(* IEC 61131-3 sources: Industry-PLC-LLM/data/PLCBEAD_repo/PLCBEAD_PLCEmbed-main/PLC-BEAD/Source/OpenPLCv2 (part 6) *)

(* ---- INC_DEC.ST ---- *)
FUNCTION_BLOCK INC_DEC_Block

	VAR_INPUT
		CHA :	BOOL;
		CHB :	BOOL;
		RST :	BOOL := 0;
	END_VAR

	VAR_OUTPUT
		DIR :	BOOL;
		CNT :	INT;
	END_VAR

	VAR
		edgea :	BOOL := 0;
		clk :	BOOL;
		clka :	BOOL;
		clkb :	BOOL;
		edgeb :	BOOL;
		axb :	BOOL;
	END_VAR

	axb := cha XOR chb;

	clka := cha XOR edgea;
	edgea := cha;

	clkb := chb XOR edgeb;
	edgeb := chb;

	clk := clka OR clkb;

	IF axb AND clka THEN dir := TRUE; END_IF;
	IF axb AND clkb THEN dir := FALSE; END_IF;

	IF clk AND dir THEN cnt := cnt + 1; END_IF;
	IF clk AND NOT dir THEN cnt := cnt -1; END_IF;

	IF rst THEN cnt := 0; END_IF;

END_FUNCTION_BLOCK

PROGRAM program0

	VAR
		CHA :	BOOL;
		CHB :	BOOL;
		RST :	BOOL := 0;

		DIR :	BOOL;
		CNT :	INT;
		func_block : INC_DEC_Block;
	END_VAR
	func_block.CHA := CHA;
	func_block.CHB := CHB;
	func_block.RST := RST;
	func_block();
	DIR := func_block.DIR;
	CNT := func_block.CNT;

END_PROGRAM

CONFIGURATION Config0

	RESOURCE Res0 ON PLC
		TASK task0(INTERVAL := T#20ms,PRIORITY := 0);
		PROGRAM instance0 WITH task0 : program0;
	END_RESOURCE

END_CONFIGURATION

(* ---- INSERT250.ST ---- *)
TYPE
	oscat_STRING250             : STRING;
END_TYPE

FUNCTION_BLOCK _INSERT250
    VAR_INPUT
        IN1 :	oscat_STRING250;
        IN2 :	oscat_STRING250;
        P :	INT;
    END_VAR
    VAR_OUTPUT
        _INSERT :	oscat_STRING250;
    END_VAR
    VAR
        size :	INT;
    END_VAR

    size := LEN(IN1);
    IF size + LEN(IN2) <= 250 THEN
        P := LIMIT(0,P,size);
        IF P = 0 THEN
            _INSERT := CONCAT(IN2,IN1);
        ELSE
            _INSERT := INSERT(IN1, IN2, P);
        END_IF;
    END_IF;

END_FUNCTION_BLOCK

PROGRAM program0
	VAR
	    LocalVar1 : oscat_STRING250;
        LocalVar2 : oscat_STRING250;
        LocalVar3 : INT;
		LocalOUT  : oscat_STRING250;
		func_block : _INSERT250;
  	END_VAR
	func_block.IN1 := LocalVar1;
    func_block.IN2 := LocalVar2;
    func_block.P := LocalVar3;
	func_block();
	LocalOUT := func_block._INSERT;
END_PROGRAM

CONFIGURATION Config0
  	RESOURCE Res0 ON PLC
    	TASK task0(INTERVAL := T#20ms,PRIORITY := 0);
    	PROGRAM instance0 WITH task0 : program0;
  	END_RESOURCE
END_CONFIGURATION

(* ---- INTEGRATE.ST ---- *)
FUNCTION_BLOCK T_PLC_MS_block
	VAR_OUTPUT
		T_PLC_MS :	UDINT;
	END_VAR

	VAR_EXTERNAL
		PLC_TICKS_PER_SEC :	INT;
		PLC_SYS_TICK_CNT :	DINT;
	END_VAR

	VAR
		debug :	BOOL;(*Debug-Mode ON / OFF*)
		N :	INT;(*Debug-Faktor*)
		Offset :	UDINT;(*Debug-Offset*)
		temp :	DWORD := DWORD#1;(*Debug-Offset*)
		mode :	BOOL;(*modus*)
		faktor :	UDINT;(*Systemtakt-Faktor*)
		init :	BOOL;
		v_plc_ticks_per_sec :	UDINT;
		base :	UDINT := UDINT#1000;
	END_VAR

	IF init = FALSE THEN
		v_plc_ticks_per_sec := INT_TO_UDINT(PLC_TICKS_PER_SEC);
		IF v_plc_ticks_per_sec = UDINT#1024 THEN
			faktor := UDINT#1;
			mode := FALSE;
		ELSIF v_plc_ticks_per_sec > UDINT#0 THEN
			IF v_plc_ticks_per_sec <= base THEN
				faktor := base / v_plc_ticks_per_sec;
				mode := FALSE;
			ELSE
				faktor := v_plc_ticks_per_sec / base;
				mode := TRUE;
			END_IF;
		ELSE
			faktor := UDINT#1;
		END_IF;
		init := TRUE;
	END_IF;

	IF mode THEN
		T_PLC_MS := DINT_TO_UDINT(PLC_SYS_TICK_CNT) / faktor;
	ELSE
		T_PLC_MS := DINT_TO_UDINT(PLC_SYS_TICK_CNT) * faktor;
	END_IF;

	IF debug THEN
		T_PLC_MS := (DWORD_TO_UDINT(SHL(UDINT_TO_DWORD(T_PLC_MS),N) OR SHL(temp,N)) - UDINT#1) + Offset;
	END_IF;
END_FUNCTION_BLOCK

FUNCTION_BLOCK INTEGRATE

	VAR_INPUT
		E :	BOOL := TRUE;
		X :	REAL;
		K :	REAL := 1.0;
	END_VAR

	VAR_IN_OUT
		Y :	REAL;
	END_VAR

	VAR
		X_last :	REAL;
		init :	BOOL;
		T_PLC_MS :	T_PLC_MS_block;
		last :	UDINT;
		tx :	UDINT;
	END_VAR

	T_PLC_MS();
	tx:= T_PLC_MS.T_PLC_MS;

	IF NOT init THEN
		init := TRUE;
		X_last := X;
	ELSIF E THEN
		Y := (X + X_LAST) * 0.5E-3 * UDINT_TO_REAL(tx-last) * K + Y;
		X_last := X;
	END_IF;
	last := tx;

END_FUNCTION_BLOCK

PROGRAM program0
  VAR
	E :	BOOL := TRUE;
	X :	REAL;
	K :	REAL := 1.0;

	Y :	REAL;

	func_block : INTEGRATE;
  END_VAR
	func_block.E:=E;
	func_block.X:=X;
	func_block.K:=K;
	func_block.Y:=Y;
	func_block();
	Y:= func_block.Y;
END_PROGRAM

CONFIGURATION Config0
	VAR_GLOBAL
		PLC_TICKS_PER_SEC :	INT;
		PLC_SYS_TICK_CNT :	DINT;
	END_VAR
	RESOURCE Res0 ON PLC
		TASK task0(INTERVAL := T#20ms,PRIORITY := 0);
		PROGRAM instance0 WITH task0 : program0;
	END_RESOURCE
END_CONFIGURATION

(* ---- INTERLOCK.ST ---- *)
FUNCTION_BLOCK INTERLOCK_Block

	VAR_INPUT
		I1 :	BOOL;
		I2 :	BOOL;
		TL :	TIME;
	END_VAR

	VAR_OUTPUT
		Q1 :	BOOL;
		Q2 :	BOOL;
	END_VAR

	VAR
		T1 :	TOF;
		T2 :	TOF;
	END_VAR

	T1(IN := I1, PT := TL);
	T2(IN := I2, PT := TL);

	Q1 := I1 AND NOT t2.Q;
	Q2 := I2 AND NOT t1.Q;

END_FUNCTION_BLOCK

PROGRAM program0
	VAR
		I1 :	BOOL;
		I2 :	BOOL;
		TL :	TIME;
		Q1 :	BOOL;
		Q2 :	BOOL;
		func_block : INTERLOCK_Block;
  	END_VAR
	func_block.I1  :=I1;
	func_block.I2  :=I2;
	func_block.TL  :=TL;
	func_block();
	Q1 := func_block.Q1;
	Q2 := func_block.Q2;
END_PROGRAM

CONFIGURATION Config0
	RESOURCE Res0 ON PLC
		TASK task0(INTERVAL := T#20ms,PRIORITY := 0);
		PROGRAM instance0 WITH task0 : program0;
	END_RESOURCE
END_CONFIGURATION

(* ---- INTERLOCK_4.ST ---- *)
FUNCTION BIT_LOAD_B:BYTE
	VAR_INPUT
		IN :	BYTE;
		VAL :	BOOL;
		POS :	INT;
	END_VAR

	IF VAL THEN
		BIT_LOAD_B := in OR SHL(BYTE#1,pos);
	ELSE
		BIT_LOAD_B := in AND (NOT SHL(BYTE#1,pos));
	END_IF;
END_FUNCTION

FUNCTION_BLOCK INTERLOCK_4_Block

	VAR_INPUT
		I0 :	BOOL;
		I1 :	BOOL;
		I2 :	BOOL;
		I3 :	BOOL;
		E :	BOOL;
		MODE :	INT;
	END_VAR

	VAR_OUTPUT
		OUT :	BYTE;
		_TP :	BOOL;
	END_VAR

	VAR
		in :	BYTE;
		last :	BYTE;
		old :	BYTE;
		lmode :	INT;
	END_VAR

	IF E THEN
	(* reset all vars when there is a mode change on thy fly *)
		IF mode <> lmode THEN
			out := BYTE#0;
			last := BYTE#0;
			old := BYTE#0;
			lmode := mode;
		END_IF;
		(* load inputs into in *)
		in:=BIT_LOAD_B(in,I0,0); (* in.0 *)
		in:=BIT_LOAD_B(in,I1,1); (* in.1 *)
		in:=BIT_LOAD_B(in,I2,2); (* in.2 *)
		in:=BIT_LOAD_B(in,I3,3); (* in.3 *)
		(* only execute when there is any change *)
		IF in <> last THEN
			(* only execute when inputs have chages state *)
			CASE mode OF
				0:	(* output directly display inputs as bits in byte out *)
					out := in;

				1:	(* the input with the highest number will be acepted *)
					IF    (in AND BYTE#2#00001000) > BYTE#0 (* in.3 *) THEN out := BYTE#8;
					ELSIF (in AND BYTE#2#00000100) > BYTE#0 (* in.2 *) THEN out := BYTE#4;
					ELSIF (in AND BYTE#2#00000010) > BYTE#0 (* in.1 *) THEN out := BYTE#2;
					ELSE out := in;
					END_IF;

				2:	(* input last pressed will be displayed only *)
					last := ((in XOR last) AND in);
					IF    (last AND BYTE#2#00001000) > BYTE#0 (* last.3 *) THEN out := BYTE#8;
					ELSIF (last AND BYTE#2#00000100) > BYTE#0 (* last.2 *) THEN out := BYTE#4;
					ELSIF (last AND BYTE#2#00000010) > BYTE#0 (* last.1 *) THEN out := BYTE#2;
					ELSE out := last;
					END_IF;

				3:	(* any input active will disable all other inputs *)
					IF (out AND in) = BYTE#0 THEN
						IF    (in AND BYTE#2#00001000) > BYTE#0 (* in.3 *) THEN out := BYTE#8;
						ELSIF (in AND BYTE#2#00000100) > BYTE#0 (* in.2 *) THEN out := BYTE#4;
						ELSIF (in AND BYTE#2#00000010) > BYTE#0 (* in.1 *) THEN out := BYTE#2;
						ELSE out := in;
						END_IF;
					END_IF;

			END_CASE;
			last := in;
		END_IF;
		_tp := out <> old;
		old := out;
	ELSE
		out := BYTE#0;
		last := BYTE#0;
		old := BYTE#0;
		lmode := 0;
		_tp := FALSE;
	END_IF;

END_FUNCTION_BLOCK

PROGRAM program0

	VAR
		I0 :	BOOL;
		I1 :	BOOL;
		I2 :	BOOL;
		I3 :	BOOL;
		E :	BOOL;
		MODE :	INT;
		OUT :	BYTE;
		_TP :	BOOL;
		func_block : INTERLOCK_4_Block;
	END_VAR
	func_block.I0 := I0;
	func_block.I1 := I1;
	func_block.I2 := I2;
	func_block.I3 := I3;
	func_block.E := E;
	func_block.MODE := MODE;
	func_block();
	OUT := func_block.OUT;
	_TP := func_block._TP;

END_PROGRAM

CONFIGURATION Config0

	RESOURCE Res0 ON PLC
		TASK task0(INTERVAL := T#20ms,PRIORITY := 0);
		PROGRAM instance0 WITH task0 : program0;
	END_RESOURCE

END_CONFIGURATION

(* ---- IP4_TO_STRING.ST ---- *)
TYPE
  oscat_STRING10             : STRING;
END_TYPE

FUNCTION _BYTE_TO_INT:INT
	VAR_INPUT
		IN :	BYTE;
	END_VAR

	_BYTE_TO_INT := USINT_TO_INT(BYTE_TO_USINT(IN));
END_FUNCTION

FUNCTION BYTE_OF_DWORD:BYTE
	VAR_INPUT
		IN :	DWORD;
		N :	BYTE;
	END_VAR
	BYTE_OF_DWORD := DWORD_TO_BYTE(SHR(in,_BYTE_TO_INT(SHL(n,3))));
END_FUNCTION

FUNCTION_BLOCK IP4_TO_STRING_Block

	VAR_INPUT
		IP4 :	DWORD;
	END_VAR

	VAR_OUTPUT
		IP4_TO_STRING :	STRING;
	END_VAR

	VAR
		s1 :	oscat_string10;
		s2 :	oscat_string10;
	END_VAR

	s1 := CONCAT(BYTE_TO_STRING(BYTE_OF_DWORD(IP4,BYTE#1)),BYTE_TO_STRING(BYTE_OF_DWORD(IP4,BYTE#0)));
	s2 := CONCAT(BYTE_TO_STRING(BYTE_OF_DWORD(IP4,BYTE#3)),BYTE_TO_STRING(BYTE_OF_DWORD(IP4,BYTE#2)));
	IP4_TO_STRING := CONCAT(s2,s1);

END_FUNCTION_BLOCK

PROGRAM program0
	VAR
		IP4 :	DWORD;
		IP4_TO_STRING :	STRING;

		func_block : IP4_TO_STRING_Block;
	END_VAR
	func_block.IP4 := IP4;

	func_block();
	IP4_TO_STRING  := func_block.IP4_TO_STRING;
END_PROGRAM

CONFIGURATION Config0

  	RESOURCE Res0 ON PLC
    	TASK task0(INTERVAL := T#20ms,PRIORITY := 0);
    	PROGRAM instance0 WITH task0 : program0;
  	END_RESOURCE

END_CONFIGURATION

(* ---- IRTRANS_DECODE.ST ---- *)
FUNCTION_BLOCK CHR_TO_STRING_Block
	VAR_INPUT
		C :	BYTE;
	END_VAR

	VAR_OUTPUT
		CHR_TO_STRING :	STRING;
	END_VAR

	CHR_TO_STRING := BYTE_TO_STRING(C);

END_FUNCTION_BLOCK

TYPE

  oscat_NW_BUF_SHORT : ARRAY [0..1407] OF BYTE;
  oscat_NW_BUF_LONG  : ARRAY [0..4095] OF BYTE;

  oscat_NETWORK_BUFFER_SHORT :
  STRUCT
    SIZE   : UINT;
    BUFFER : oscat_NW_BUF_SHORT;
  END_STRUCT;

  oscat_NETWORK_BUFFER :
  STRUCT
    SIZE   : UINT;
    BUFFER : oscat_NW_BUF_LONG;
  END_STRUCT;

END_TYPE

TYPE
  oscat_IP_FIFO128_DATA  : ARRAY [1..128] OF BYTE;
  oscat_Mailbox  : ARRAY [1..16] OF BYTE;

  oscat_IP_FIFO_DATA :
  STRUCT
	X       : oscat_IP_FIFO128_DATA; (* IP_ID FIFO Speicher          *)
	Y       : oscat_IP_FIFO128_DATA; (* IP_ID Z�hler                 *)
	ID      : BYTE;                  (* h�chste vergabene id         *)
	MAX_ID  : BYTE;                  (* maximal Anmeldungen pro ID   *)
    INIT    : BOOL;                  (* Initialisierung durchgef�hrt *)
	EMPTY   : BOOL;                  (* FIFO leer                    *)
	FULL    : BOOL;                  (* FIFO voll                    *)
	TOP     : INT;                   (* maximale anzahl in FIFO      *)
	NW      : INT;                   (* Schreibzeiger                *)
	NR      : INT;                   (* Lesezeiger                   *)
  END_STRUCT;

  oscat_IP_C:
  STRUCT
  	C_MODE:			BYTE;          		(*W Mode: TCP/UCP AKTIV/PASSIV                               *)
	C_PORT:         WORD;          		(*W Portnummer                                               *)
	C_IP:           DWORD;         		(*W IP-Adresse gepackt wwxxyyzz = www.xxx.yyy.zzz            *)
    C_STATE:        BYTE;          		(*R Verbindungsstatus ON/OFF + Flanke ON/OFF                 *)
	C_ENABLE:       BOOL;          		(*W Freigabe f�r Connect                                     *)
    R_OBSERVE:      BOOL;          		(*W Empfang ueberwachen                                      *)
    TIME_RESET:     BOOL;          		(*W Alle Timer ruecksetzen                                   *)
	ERROR:          DWORD;         		(*R vvwwxxyy (vv = CON_ERROR, ww = SEN_ERROR, xx = REC_ERROR *)
    FIFO:           oscat_IP_FIFO_DATA; (*I IP FIFO Struktur                                         *)
	MAILBOX:		oscat_Mailbox;		(*I Mailbox: Datenbereich f�r Bausteindatenaustausch         *)
  END_STRUCT;
END_TYPE

FUNCTION_BLOCK IRTRANS_DECODE_Block

	VAR_OUTPUT
		CMD :	BOOL;
		DEV :	STRING;
		KEY :	STRING;
		ERROR :	BOOL;
	END_VAR

	VAR_IN_OUT
		IP_C :	oscat_IP_C;
		R_BUF :	oscat_NETWORK_BUFFER;
	END_VAR

	VAR
		i :	INT;
		stop :	INT;
		received_string :	STRING;
		char :	STRING;
		CHR_TO_STRING :	CHR_TO_STRING_Block;
		z :	BYTE;
	END_VAR

	i := UINT_TO_INT(R_BUF.SIZE);
	IF i >= 5 AND (i <= 82) AND IP_C.MAILBOX[1] <> z THEN
		error := TRUE;
		i := i - 1;

		IF R_BUF.BUFFER[i] <> BYTE#10 THEN RETURN; END_IF;
		i := i - 1;
		IF R_BUF.BUFFER[i] <> BYTE#13 THEN RETURN; END_IF;
		i := i - 1;

		stop := 0;
		received_string := '';

		WHILE stop <= i DO
			CHR_TO_STRING(C:=R_BUF.BUFFER[stop]);
			char := CHR_TO_STRING.CHR_TO_STRING;
			received_string := CONCAT(received_string,char);
			stop := stop + INT#1;
		END_WHILE;

		stop := FIND(received_string,',');
		IF stop > 0 AND stop - 1 < i THEN
			DEV := LEFT(received_string,stop - 1);
			key := RIGHT(received_string,i - stop + 1);
			IF LEN(DEV) = 0 OR LEN(key) = 0 THEN RETURN; END_IF;
			cmd := TRUE;
			error := FALSE;
		END_IF;
	ELSE
		cmd := FALSE;
		error := FALSE;
	END_IF;

	z := IP_C.MAILBOX[1];

END_FUNCTION_BLOCK

PROGRAM program0
	VAR
		IP_C :	oscat_IP_C;
		R_BUF :	oscat_NETWORK_BUFFER;
		CMD :	BOOL;
		DEV :	STRING;
		KEY :	STRING;
		ERROR :	BOOL;

		func_block : IRTRANS_DECODE_Block;
	END_VAR
	func_block.IP_C := IP_C;
	func_block.R_BUF := R_BUF;

	func_block();
	IP_C  := func_block.IP_C;
	R_BUF  := func_block.R_BUF;
	CMD  := func_block.CMD;
	DEV  := func_block.DEV;
	KEY  := func_block.KEY;
	ERROR  := func_block.ERROR;

END_PROGRAM

CONFIGURATION Config0

  	RESOURCE Res0 ON PLC
    	TASK task0(INTERVAL := T#20ms,PRIORITY := 0);
    	PROGRAM instance0 WITH task0 : program0;
  	END_RESOURCE

END_CONFIGURATION

(* ---- IRTRANS_RCV_1.ST ---- *)
FUNCTION_BLOCK IRTRANS_RCV_1_Block

	VAR_INPUT
		CMD :	BOOL;
		DEV_CODE :	STRING;
		KEY_CODE :	STRING;
	END_VAR

	VAR_OUTPUT
		Q :	BOOL;
	END_VAR

	VAR_IN_OUT
		DEV :	STRING;
		KEY :	STRING;
	END_VAR

	Q := cmd AND EQ_STRING(dev_code,dev) AND EQ_STRING(key_code,key);

END_FUNCTION_BLOCK

PROGRAM program0
	VAR
		CMD :	BOOL;
		DEV :	STRING;
		KEY :	STRING;
		DEV_CODE :	STRING;
		KEY_CODE :	STRING;
		Q :	BOOL;

		func_block : IRTRANS_RCV_1_Block;
	END_VAR
	func_block.CMD := CMD;
	func_block.DEV := DEV;
	func_block.KEY := KEY;
	func_block.DEV_CODE := DEV_CODE;
	func_block.KEY_CODE := KEY_CODE;

	func_block();
	DEV  := func_block.DEV;
	KEY  := func_block.KEY;
	Q  := func_block.Q;

END_PROGRAM

CONFIGURATION Config0

  	RESOURCE Res0 ON PLC
    	TASK task0(INTERVAL := T#20ms,PRIORITY := 0);
    	PROGRAM instance0 WITH task0 : program0;
  	END_RESOURCE

END_CONFIGURATION

(* ---- IRTRANS_RCV_4.ST ---- *)
FUNCTION_BLOCK IRTRANS_RCV_4_Block

	VAR_INPUT
		CMD :	BOOL;
	END_VAR

	VAR_IN_OUT
		DEV :	STRING;
		KEY :	STRING;
	END_VAR

	VAR_INPUT
		DEV_CODE :	STRING;
		KEY_CODE_0 :	STRING;
		KEY_CODE_1 :	STRING;
		KEY_CODE_2 :	STRING;
		KEY_CODE_3 :	STRING;
	END_VAR

	VAR_OUTPUT
		Q0 :	BOOL;
		Q1 :	BOOL;
		Q2 :	BOOL;
		Q3 :	BOOL;
	END_VAR

	VAR
		decode :	BOOL;
	END_VAR

	decode := cmd AND EQ_STRING(dev_code,dev);

	Q0 := EQ_STRING(key,key_code_0) AND decode;
	Q1 := EQ_STRING(key,key_code_1) AND decode;
	Q2 := EQ_STRING(key,key_code_2) AND decode;
	Q3 := EQ_STRING(key,key_code_3) AND decode;

END_FUNCTION_BLOCK

PROGRAM program0
	VAR
		CMD :	BOOL;
		DEV :	STRING;
		KEY :	STRING;
		DEV_CODE :	STRING;
		KEY_CODE_0 :	STRING;
		KEY_CODE_1 :	STRING;
		KEY_CODE_2 :	STRING;
		KEY_CODE_3 :	STRING;
		Q0 :	BOOL;
		Q1 :	BOOL;
		Q2 :	BOOL;
		Q3 :	BOOL;

		func_block : IRTRANS_RCV_4_Block;
	END_VAR
	func_block.CMD := CMD;
	func_block.DEV := DEV;
	func_block.KEY := KEY;
	func_block.DEV_CODE := DEV_CODE;
	func_block.KEY_CODE_0 := KEY_CODE_0;
	func_block.KEY_CODE_1 := KEY_CODE_1;
	func_block.KEY_CODE_2 := KEY_CODE_2;
	func_block.KEY_CODE_3 := KEY_CODE_3;

	func_block();
	DEV  := func_block.DEV;
	KEY  := func_block.KEY;
	Q0  := func_block.Q0;
	Q1  := func_block.Q1;
	Q2  := func_block.Q2;
	Q3  := func_block.Q3;

END_PROGRAM

CONFIGURATION Config0

  	RESOURCE Res0 ON PLC
    	TASK task0(INTERVAL := T#20ms,PRIORITY := 0);
    	PROGRAM instance0 WITH task0 : program0;
  	END_RESOURCE

END_CONFIGURATION

(* ---- IRTRANS_RCV_8.ST ---- *)
FUNCTION_BLOCK IRTRANS_RCV_8_Block

	VAR_INPUT
		CMD :	BOOL;
	END_VAR

	VAR_IN_OUT
		DEV :	STRING;
		KEY :	STRING;
	END_VAR

	VAR_INPUT
		DEV_CODE :	STRING;
		KEY_CODE_0 :	STRING;
		KEY_CODE_1 :	STRING;
		KEY_CODE_2 :	STRING;
		KEY_CODE_3 :	STRING;
		KEY_CODE_4 :	STRING;
		KEY_CODE_5 :	STRING;
		KEY_CODE_6 :	STRING;
		KEY_CODE_7 :	STRING;
	END_VAR

	VAR_OUTPUT
		Q0 :	BOOL;
		Q1 :	BOOL;
		Q2 :	BOOL;
		Q3 :	BOOL;
		Q4 :	BOOL;
		Q5 :	BOOL;
		Q6 :	BOOL;
		Q7 :	BOOL;
	END_VAR

	VAR
		decode :	BOOL;
	END_VAR

	decode := cmd AND EQ_STRING(dev_code,dev);

	Q0 := EQ_STRING(key,key_code_0) AND decode;
	Q1 := EQ_STRING(key,key_code_1) AND decode;
	Q2 := EQ_STRING(key,key_code_2) AND decode;
	Q3 := EQ_STRING(key,key_code_3) AND decode;
	Q4 := EQ_STRING(key,key_code_4) AND decode;
	Q5 := EQ_STRING(key,key_code_5) AND decode;
	Q6 := EQ_STRING(key,key_code_6) AND decode;
	Q7 := EQ_STRING(key,key_code_7) AND decode;

END_FUNCTION_BLOCK

PROGRAM program0
	VAR
		CMD :	BOOL;
		DEV :	STRING;
		KEY :	STRING;
		DEV_CODE :	STRING;
		KEY_CODE_0 :	STRING;
		KEY_CODE_1 :	STRING;
		KEY_CODE_2 :	STRING;
		KEY_CODE_3 :	STRING;
		KEY_CODE_4 :	STRING;
		KEY_CODE_5 :	STRING;
		KEY_CODE_6 :	STRING;
		KEY_CODE_7 :	STRING;
		Q0 :	BOOL;
		Q1 :	BOOL;
		Q2 :	BOOL;
		Q3 :	BOOL;
		Q4 :	BOOL;
		Q5 :	BOOL;
		Q6 :	BOOL;
		Q7 :	BOOL;

		func_block : IRTRANS_RCV_8_Block;
	END_VAR
	func_block.CMD := CMD;
	func_block.DEV := DEV;
	func_block.KEY := KEY;
	func_block.DEV_CODE := DEV_CODE;
	func_block.KEY_CODE_0 := KEY_CODE_0;
	func_block.KEY_CODE_1 := KEY_CODE_1;
	func_block.KEY_CODE_2 := KEY_CODE_2;
	func_block.KEY_CODE_3 := KEY_CODE_3;
	func_block.KEY_CODE_4 := KEY_CODE_4;
	func_block.KEY_CODE_5 := KEY_CODE_5;
	func_block.KEY_CODE_6 := KEY_CODE_6;
	func_block.KEY_CODE_7 := KEY_CODE_7;

	func_block();
	DEV  := func_block.DEV;
	KEY  := func_block.KEY;
	Q0  := func_block.Q0;
	Q1  := func_block.Q1;
	Q2  := func_block.Q2;
	Q3  := func_block.Q3;
	Q4  := func_block.Q4;
	Q5  := func_block.Q5;
	Q6  := func_block.Q6;
	Q7  := func_block.Q7;

END_PROGRAM

CONFIGURATION Config0

  	RESOURCE Res0 ON PLC
    	TASK task0(INTERVAL := T#20ms,PRIORITY := 0);
    	PROGRAM instance0 WITH task0 : program0;
  	END_RESOURCE

END_CONFIGURATION

(* ---- IRTRANS_SERVER.ST ---- *)
TYPE

  oscat_NW_BUF_SHORT : ARRAY [0..1407] OF BYTE;
  oscat_NW_BUF_LONG  : ARRAY [0..4095] OF BYTE;

  oscat_NETWORK_BUFFER_SHORT :
  STRUCT
    SIZE   : UINT;
    BUFFER : oscat_NW_BUF_SHORT;
  END_STRUCT;

  oscat_NETWORK_BUFFER :
  STRUCT
    SIZE   : UINT;
    BUFFER : oscat_NW_BUF_LONG;
  END_STRUCT;

END_TYPE

TYPE
  oscat_IP_FIFO128_DATA  : ARRAY [1..128] OF BYTE;
  oscat_Mailbox  : ARRAY [1..16] OF BYTE;

  oscat_IP_FIFO_DATA :
  STRUCT
	X       : oscat_IP_FIFO128_DATA; (* IP_ID FIFO Speicher          *)
	Y       : oscat_IP_FIFO128_DATA; (* IP_ID Z�hler                 *)
	ID      : BYTE;                  (* h�chste vergabene id         *)
	MAX_ID  : BYTE;                  (* maximal Anmeldungen pro ID   *)
    INIT    : BOOL;                  (* Initialisierung durchgef�hrt *)
	EMPTY   : BOOL;                  (* FIFO leer                    *)
	FULL    : BOOL;                  (* FIFO voll                    *)
	TOP     : INT;                   (* maximale anzahl in FIFO      *)
	NW      : INT;                   (* Schreibzeiger                *)
	NR      : INT;                   (* Lesezeiger                   *)
  END_STRUCT;

  oscat_IP_C:
  STRUCT
  	C_MODE:			BYTE;          		(*W Mode: TCP/UCP AKTIV/PASSIV                               *)
	C_PORT:         WORD;          		(*W Portnummer                                               *)
	C_IP:           DWORD;         		(*W IP-Adresse gepackt wwxxyyzz = www.xxx.yyy.zzz            *)
    C_STATE:        BYTE;          		(*R Verbindungsstatus ON/OFF + Flanke ON/OFF                 *)
	C_ENABLE:       BOOL;          		(*W Freigabe f�r Connect                                     *)
    R_OBSERVE:      BOOL;          		(*W Empfang ueberwachen                                      *)
    TIME_RESET:     BOOL;          		(*W Alle Timer ruecksetzen                                   *)
	ERROR:          DWORD;         		(*R vvwwxxyy (vv = CON_ERROR, ww = SEN_ERROR, xx = REC_ERROR *)
    FIFO:           oscat_IP_FIFO_DATA; (*I IP FIFO Struktur                                         *)
	MAILBOX:		oscat_Mailbox;		(*I Mailbox: Datenbereich f�r Bausteindatenaustausch         *)
  END_STRUCT;
END_TYPE

FUNCTION_BLOCK IRTRANS_SERVER_Block

	VAR_INPUT
		UDP_TCP :	BOOL;
	END_VAR

	VAR_OUTPUT
		S_ENABLE :	BOOL;
		R_ENABLE :	BOOL;
		ERROR :	DWORD;
	END_VAR

	VAR_IN_OUT
		IP_C :	oscat_IP_C;
		S_BUF :	oscat_NETWORK_BUFFER;
		R_BUF :	oscat_NETWORK_BUFFER;
	END_VAR

	VAR
		t :	TON;
	END_VAR

	IF NOT IP_C.C_ENABLE THEN
		IP_C.C_PORT := WORD#0;
		IP_C.C_IP := DWORD#00;
		IP_C.C_MODE := SEL(UDP_TCP,BYTE#5,BYTE#4);
		IP_C.C_ENABLE := TRUE;
		IP_C.R_OBSERVE := FALSE;
		IP_C.TIME_RESET := TRUE;
		S_BUF.SIZE := UINT#0;
		R_BUF.SIZE := UINT#0;
	END_IF;

	R_ENABLE := IP_C.C_STATE > BYTE#127;
	S_ENABLE := R_ENABLE AND (IP_C.MAILBOX[1] > BYTE#0 OR IP_C.C_MODE <> BYTE#5);
	ERROR := IP_C.ERROR;

	t(IN:= IP_C.ERROR > DWORD#0, PT:=T#5s);
	IF t.Q THEN
		IP_C.TIME_RESET := TRUE;
	END_IF;

END_FUNCTION_BLOCK

PROGRAM program0
	VAR
		UDP_TCP :	BOOL;
		S_ENABLE :	BOOL;
		R_ENABLE :	BOOL;
		ERROR :	DWORD;
		IP_C :	oscat_IP_C;
		S_BUF :	oscat_NETWORK_BUFFER;
		R_BUF :	oscat_NETWORK_BUFFER;

		func_block : IRTRANS_SERVER_Block;
	END_VAR
	func_block.UDP_TCP := UDP_TCP;
	func_block.IP_C := IP_C;
	func_block.S_BUF := S_BUF;
	func_block.R_BUF := R_BUF;

	func_block();
	S_ENABLE  := func_block.S_ENABLE;
	R_ENABLE  := func_block.R_ENABLE;
	ERROR  := func_block.ERROR;
	IP_C  := func_block.IP_C;
	S_BUF  := func_block.S_BUF;
	R_BUF  := func_block.R_BUF;

END_PROGRAM

CONFIGURATION Config0

  	RESOURCE Res0 ON PLC
    	TASK task0(INTERVAL := T#20ms,PRIORITY := 0);
    	PROGRAM instance0 WITH task0 : program0;
  	END_RESOURCE

END_CONFIGURATION

(* ---- IS_CC.ST ---- *)
FUNCTION_BLOCK IS_CC_Block

	VAR_INPUT
		STR :	STRING;
		CMP :	STRING;
	END_VAR

	VAR_OUTPUT
		IS_CC :	BOOL;
	END_VAR

	VAR
		L :	INT;
		pos :	INT;
		temp :	STRING;
	END_VAR

	L := LEN(str);
	FOR pos := 1 TO L DO
		temp := MID(str,1,pos);
		IF FIND(CMP,temp) = 0 THEN
			IS_CC := FALSE;
			RETURN;
		END_IF;
	END_FOR;
	IS_CC := L > 0;

END_FUNCTION_BLOCK

PROGRAM program0

	VAR
		STR :	STRING;
		CMP :	STRING;

		IS_CC :	BOOL;

		func_block : IS_CC_Block;
	END_VAR
	func_block.STR := STR;
	func_block.CMP := CMP;
	func_block();
	IS_CC := func_block.IS_CC;

END_PROGRAM

CONFIGURATION Config0

	RESOURCE Res0 ON PLC
		TASK task0(INTERVAL := T#20ms,PRIORITY := 0);
		PROGRAM instance0 WITH task0 : program0;
	END_RESOURCE

END_CONFIGURATION

(* ---- IS_NCC.ST ---- *)
FUNCTION_BLOCK IS_NCC_Block

	VAR_INPUT
		STR :	STRING;
		CMP :	STRING;
	END_VAR

	VAR_OUTPUT
		IS_NCC :	BOOL;
	END_VAR

	VAR
		L :	INT;
		pos :	INT;
		temp :	STRING;
	END_VAR

	L := LEN(str);
	FOR pos := 1 TO L DO
		temp := MID(str,1,pos);
		IF FIND(CMP,temp) > 0 THEN
			IS_NCC := FALSE;
			RETURN;
		END_IF;
	END_FOR;
	IS_NCC := TRUE;

END_FUNCTION_BLOCK

PROGRAM program0

	VAR
		STR :	STRING;
		CMP :	STRING;
		IS_NCC :	BOOL;
		func_block : IS_NCC_Block;
	END_VAR
	func_block.STR := STR;
	func_block.CMP := CMP;
	func_block();
	IS_NCC := func_block.IS_NCC;

END_PROGRAM

CONFIGURATION Config0

	RESOURCE Res0 ON PLC
		TASK task0(INTERVAL := T#20ms,PRIORITY := 0);
		PROGRAM instance0 WITH task0 : program0;
	END_RESOURCE

END_CONFIGURATION

(* ---- IS_SORTED.ST ---- *)
TYPE
	oscat_pt_ARRAY: ARRAY [1..100] OF REAL;
END_TYPE

FUNCTION_BLOCK IS_SORTED_Block

	VAR_IN_OUT
		PT :	oscat_pt_ARRAY;
	END_VAR

	VAR_INPUT
		SIZE :	UINT;
	END_VAR

	VAR_OUTPUT
		IS_SORTED :	BOOL;
	END_VAR

	VAR
		i :	INT;
		i2 :	INT;
		stop :	INT;
	END_VAR

	stop :=LIMIT_INT(1,UINT_TO_INT(size),1000);
	stop := stop -1;
	FOR i := 1 TO stop DO
		i2 := i+1;
		IF pt[i] > pt[i2] THEN
			IS_SORTED := FALSE;
			RETURN;
		END_IF;
	END_FOR;

	IS_SORTED := TRUE;

END_FUNCTION_BLOCK

PROGRAM program0

	VAR
		SIZE :	UINT;
		PT :	oscat_pt_ARRAY;
		IS_SORTED :	BOOL;
		func_block : IS_SORTED_Block;
	END_VAR
	func_block.SIZE := SIZE;
	func_block.PT := PT;
	func_block();
	PT := func_block.PT;
	IS_SORTED := func_block.IS_SORTED;

END_PROGRAM

CONFIGURATION Config0

	RESOURCE Res0 ON PLC
		TASK task0(INTERVAL := T#20ms,PRIORITY := 0);
		PROGRAM instance0 WITH task0 : program0;
	END_RESOURCE

END_CONFIGURATION

(* ---- LAMBERT_W.ST ---- *)
FUNCTION _REAL_TO_DWORD: DWORD

  VAR_INPUT
    X :	REAL;
  END_VAR

  IF REAL_TO_DWORD(0.5) = DWORD#1 THEN
    _REAL_TO_DWORD := REAL_TO_DWORD(x);
  ELSIF X > 0.0 THEN
    _REAL_TO_DWORD := REAL_TO_DWORD(x+0.5);
  ELSIF X < 0.0 THEN
    _REAL_TO_DWORD := REAL_TO_DWORD(x-0.5);
  ELSE
    _REAL_TO_DWORD := DWORD#0;
  END_IF;
END_FUNCTION

FUNCTION_BLOCK LAMBERT_W_Block

	VAR_INPUT
		X :	REAL;
	END_VAR

	VAR_OUTPUT
		LAMBERT_W :	REAL;
	END_VAR

	VAR
		w :	REAL;
		i :	INT;
		we :	REAL;
		w1e :	REAL;
		last :	DWORD;
		ewx :	REAL;
	END_VAR

	IF x < -0.367879441171442 THEN
		LAMBERT_W := -1000.0;
		RETURN;
	(* return 0 if x = 0 *)
	ELSIF x = 0.0 THEN
		RETURN;
	(* first an estimate is calculated *)
	ELSIF x <= 500.0 THEN
		w := LN(x + 1.0);
		w := 0.665 * (1.0 + 0.0195 * w) * w + 0.04;
	ELSE
		w := LN(x - 4.0) - (1.0 - 1.0/LN(x)) * LN(LN(x));
	END_IF;
	(* use estimate to calculate exact result *)
	FOR i := 0 TO 5 DO
		ewx := EXP(w);
		we := w * ewx - x;
		w1e := (w+1.0) * ewx;
		last := _REAL_TO_DWORD(w) AND DWORD#16#FFFF_FFFC;
		w := w - (we / (w1e - (w+2.0) * we / (2.0 * w + 2.0)));
		IF (_REAL_TO_DWORD(w) AND DWORD#16#FFFF_FFFC) = last THEN EXIT; END_IF;
	END_FOR;
	LAMBERT_W := w;

END_FUNCTION_BLOCK

PROGRAM program0

	VAR
		X :	REAL;
		LAMBERT_W :	REAL;
		func_block : LAMBERT_W_Block;
	END_VAR
	func_block.X := X;
	func_block();
	LAMBERT_W := func_block.LAMBERT_W;

END_PROGRAM

CONFIGURATION Config0

	RESOURCE Res0 ON PLC
		TASK task0(INTERVAL := T#20ms,PRIORITY := 0);
		PROGRAM instance0 WITH task0 : program0;
	END_RESOURCE

END_CONFIGURATION

(* ---- LEGIONELLA.ST ---- *)
FUNCTION TIMECHECK:BOOL

	VAR_INPUT
		TD :	UDINT;
		START :	UDINT;
		STOP :	UDINT;
	END_VAR

	IF stop < start THEN
		TIMECHECK := start <= TD OR  TD < stop;
	ELSE
		TIMECHECK := start <= TD AND TD < stop;
	END_IF;

END_FUNCTION

FUNCTION TIME_TO_TOD:UDINT

	VAR_INPUT
		IN :	TIME;
	END_VAR

	TIME_TO_TOD := DWORD_TO_UDINT(TIME_TO_DWORD(IN));
END_FUNCTION

FUNCTION TOD_TO_TIME:TIME
	VAR_INPUT
		IN :	UDINT;
	END_VAR

	TOD_TO_TIME := DWORD_TO_TIME(UDINT_TO_DWORD(IN));
END_FUNCTION

FUNCTION DAY_OF_WEEK:INT
  VAR_INPUT
    IDATE :	UDINT;
  END_VAR

  DAY_OF_WEEK := UDINT_TO_INT((idate / UDINT#86400 + UDINT#3) MOD UDINT#7) + INT#01;
END_FUNCTION

FUNCTION _DT_TO_DATE_B:UDINT

	VAR_INPUT
		_INN :	UDINT;
	END_VAR

	_DT_TO_DATE_B := (_INN / UDINT#86400) * UDINT#86400;
END_FUNCTION

FUNCTION DT_TO_TOD2:UDINT
	VAR_INPUT
		IN :	UDINT;
	END_VAR

	DT_TO_TOD2 := (IN MOD UDINT#86400) * UDINT#1000;
END_FUNCTION

FUNCTION TIME_TO_TOD2:UDINT

	VAR_INPUT
		IN :	TIME;
	END_VAR

	TIME_TO_TOD2 := DWORD_TO_UDINT(TIME_TO_DWORD(IN));
END_FUNCTION

FUNCTION_BLOCK TIMER_1_Block

	VAR_INPUT
		E :	BOOL := TRUE;
		DTI :	UDINT;
		START :	UDINT;
		DURATION :	TIME;
		DAY :	BYTE := BYTE#2#0111_1111;
	END_VAR

	VAR_OUTPUT
		Q :	BOOL;
		STOP :	TIME;
	END_VAR

	IF E THEN
		stop := TOD_TO_TIME(START) + DURATION;
		IF stop > T#24h THEN stop := stop - T#24h; END_IF;
		Q := TIMECHECK(DT_TO_TOD2(DTI), START, TIME_TO_TOD2(stop)) AND (SHR(BYTE#128, DAY_OF_WEEK(_DT_TO_DATE_B(DTI))) AND DAY) > BYTE#0;
	ELSE
		Q := FALSE;
	END_IF;

END_FUNCTION_BLOCK

FUNCTION UDINT_TO_TIME2:TIME

	VAR_INPUT
		IN :	UDINT;
	END_VAR

	UDINT_TO_TIME2 := DINT_TO_TIME(UDINT_TO_DINT(IN));

END_FUNCTION

FUNCTION_BLOCK T_PLC_MS_block
	VAR_OUTPUT
		T_PLC_MS :	UDINT;
	END_VAR

	VAR_EXTERNAL
		PLC_TICKS_PER_SEC :	INT;
		PLC_SYS_TICK_CNT :	DINT;
	END_VAR

	VAR
		debug :	BOOL;
		N :	INT;
		Offset :	UDINT;
		temp :	DWORD := DWORD#1;
		mode :	BOOL;
		faktor :	UDINT;
		init :	BOOL;
		v_plc_ticks_per_sec :	UDINT;
		base :	UDINT := UDINT#1000;
	END_VAR

	IF init = FALSE THEN
		v_plc_ticks_per_sec := INT_TO_UDINT(PLC_TICKS_PER_SEC);
		IF v_plc_ticks_per_sec = UDINT#1024 THEN
			faktor := UDINT#1;
			mode := FALSE;
		ELSIF v_plc_ticks_per_sec > UDINT#0 THEN
			IF v_plc_ticks_per_sec <= base THEN
				faktor := base / v_plc_ticks_per_sec;
				mode := FALSE;
			ELSE
				faktor := v_plc_ticks_per_sec / base;
				mode := TRUE;
			END_IF;
		ELSE
			faktor := UDINT#1;
		END_IF;
		init := TRUE;
	END_IF;

	IF mode THEN
		T_PLC_MS := DINT_TO_UDINT(PLC_SYS_TICK_CNT) / faktor;
	ELSE
		T_PLC_MS := DINT_TO_UDINT(PLC_SYS_TICK_CNT) * faktor;
	END_IF;

	IF debug THEN
		T_PLC_MS := (DWORD_TO_UDINT(SHL(UDINT_TO_DWORD(T_PLC_MS),N) OR SHL(temp,N)) - UDINT#1) + Offset;
	END_IF;

END_FUNCTION_BLOCK

FUNCTION_BLOCK SEQUENCE_8_Block

	VAR_INPUT
		IN0 :	BOOL := TRUE;
		IN1 :	BOOL := TRUE;
		IN2 :	BOOL := TRUE;
		IN3 :	BOOL := TRUE;
		IN4 :	BOOL := TRUE;
		IN5 :	BOOL := TRUE;
		IN6 :	BOOL := TRUE;
		IN7 :	BOOL := TRUE;
		START :	BOOL;
		RST :	BOOL;
		WAIT0 :	TIME;
		DELAY0 :	TIME;
		WAIT1 :	TIME;
		DELAY1 :	TIME;
		WAIT2 :	TIME;
		DELAY2 :	TIME;
		WAIT3 :	TIME;
		DELAY3 :	TIME;
		WAIT4 :	TIME;
		DELAY4 :	TIME;
		WAIT5 :	TIME;
		DELAY5 :	TIME;
		WAIT6 :	TIME;
		DELAY6 :	TIME;
		WAIT7 :	TIME;
		DELAY7 :	TIME;
		STOP_ON_ERROR :	BOOL;
	END_VAR

	VAR_OUTPUT
		Q0 :	BOOL;
		Q1 :	BOOL;
		Q2 :	BOOL;
		Q3 :	BOOL;
		Q4 :	BOOL;
		Q5 :	BOOL;
		Q6 :	BOOL;
		Q7 :	BOOL;
		QX :	BOOL;
		RUN :	BOOL;
		_STEP :	INT := -1;
		STATUS :	BYTE;
	END_VAR

	VAR
		last :	TIME;
		edge :	BOOL;
		tx :	TIME;
		init :	BOOL;
		T_PLC_MS :	T_PLC_MS_Block;
	END_VAR

	T_PLC_MS();
	tx:= UDINT_TO_TIME(T_PLC_MS.T_PLC_MS);

	IF NOT init THEN
		last := tx;
		init := TRUE;
		status := BYTE#110;
	END_IF;

	IF rst THEN
		_step := -1;
		Q0 := FALSE;
		Q1 := FALSE;
		Q2 := FALSE;
		Q3 := FALSE;
		Q4 := FALSE;
		Q5 := FALSE;
		Q6 := FALSE;
		Q7 := FALSE;
		status := BYTE#110;
		run := FALSE;

	ELSIF start AND NOT edge THEN
		_step := 0;
		last := tx;
		status := BYTE#111;
		Q0 := FALSE;
		Q1 := FALSE;
		Q2 := FALSE;
		Q3 := FALSE;
		Q4 := FALSE;
		Q5 := FALSE;
		Q6 := FALSE;
		Q7 := FALSE;
		run := TRUE;
	END_IF;
	edge := start;

	IF status > BYTE#0 AND status < BYTE#100 AND stop_on_error THEN RETURN; END_IF;

	IF run AND _step = 0 THEN
		IF NOT q0 AND in0 AND tx - last <= wait0 THEN
			Q0 := TRUE;
			last := tx;
		ELSIF NOT q0 AND tx - last > wait0 THEN
			status := BYTE#1;
			run := FALSE;
		ELSIF q0 AND tx - last >= delay0 THEN
			_step := 1;
			last := tx;
		END_IF;
	END_IF;
	IF run AND _step = 1 THEN
		IF NOT q1 AND in1 AND tx - last <= wait1 THEN
			Q0 := FALSE;
			Q1 := TRUE;
			last := tx;
		ELSIF NOT q1 AND Tx - last > wait1 THEN
			status := BYTE#2;
			q0 := FALSE;
			run := FALSE;
		ELSIF q1 AND tx - last >= delay1 THEN
			_step := 2;
			last := tx;
		END_IF;
	END_IF;
	IF run AND _step = 2 THEN
		IF NOT q2 AND in2 AND tx - last <= wait2 THEN
			Q1 := FALSE;
			Q2 := TRUE;
			last := tx;
		ELSIF NOT q2 AND Tx - last > wait2 THEN
			status := BYTE#3;
			q1 := FALSE;
			run := FALSE;
		ELSIF q2 AND tx - last >= delay2 THEN
			_step := 3;
			last := tx;
		END_IF;
	END_IF;
	IF run AND _step = 3 THEN
		IF NOT q3 AND in3 AND tx - last <= wait3 THEN
			Q2 := FALSE;
			Q3 := TRUE;
			last := tx;
		ELSIF NOT q3 AND Tx - last > wait3 THEN
			status := BYTE#4;
			q2 := FALSE;
			run := FALSE;
		ELSIF q3 AND tx - last >= delay3 THEN
			_step := 4;
			last := tx;
		END_IF;
	END_IF;
	IF run AND _step = 4 THEN
		IF NOT q4 AND in4 AND tx - last <= wait4 THEN
			Q3 := FALSE;
			Q4 := TRUE;
			last := tx;
		ELSIF NOT q4 AND Tx - last > wait4 THEN
			status := BYTE#5;
			q3 := FALSE;
			run := FALSE;
		ELSIF q4 AND tx - last >= delay4 THEN
			_step := 5;
			last := tx;
		END_IF;
	END_IF;
	IF run AND _step = 5 THEN
		IF NOT q5 AND in5 AND tx - last <= wait5 THEN
			Q4 := FALSE;
			Q5 := TRUE;
			last := tx;
		ELSIF NOT q5 AND Tx - last > wait5 THEN
			status := BYTE#6;
			q4 := FALSE;
			run := FALSE;
		ELSIF q5 AND tx - last >= delay5 THEN
			_step := 6;
			last := tx;
		END_IF;
	END_IF;
	IF run AND _step = 6 THEN
		IF NOT q6 AND in6 AND tx - last <= wait6 THEN
			Q5 := FALSE;
			Q6 := TRUE;
			last := tx;
		ELSIF NOT q6 AND Tx - last > wait6 THEN
			status := BYTE#7;
			q5 := FALSE;
			run := FALSE;
		ELSIF q6 AND tx - last >= delay6 THEN
			_step := 7;
			last := tx;
		END_IF;
	END_IF;
	IF run AND _step = 7 THEN
		IF NOT q7 AND in7 AND tx - last <= wait7 THEN
			Q6 := FALSE;
			Q7 := TRUE;
			last := tx;
		ELSIF NOT q7 AND Tx - last > wait7 THEN
			status := BYTE#8;
			q6 := FALSE;
			run := FALSE;
		ELSIF q7 AND tx - last >= delay7 THEN
			_step := -1;
			Q7 := FALSE;
			Run := FALSE;
			status := BYTE#110;
		END_IF;
	END_IF;
	QX := q0 OR q1 OR q2 OR q3 OR q4 OR q5 OR q6 OR q7;

END_FUNCTION_BLOCK

FUNCTION_BLOCK HYST_1_Block

	VAR_INPUT
		IN :	REAL;
		HIGH :	REAL;
		LOW :	REAL;
	END_VAR

	VAR_OUTPUT
		Q :	BOOL;
		WIN :	BOOL;
	END_VAR

	IF in < low THEN
		Q := FALSE;
		win := FALSE;
	ELSIF in > high THEN
		Q := TRUE;
		win := FALSE;
	ELSE
		win := TRUE;
	END_IF;

END_FUNCTION_BLOCK

FUNCTION_BLOCK LEGIONELLA_Block

	VAR_INPUT
		MANUAL :	BOOL;
		TEMP_BOILER :	REAL;
		TEMP_RETURN :	REAL := 100.0;
		DT_IN :	UDINT;
		RST :	BOOL;
		T_START :	UDINT := UDINT#10800000;(*tod#03:00:00*)
		DAY :	INT := 7;
		TEMP_SET :	REAL := 70.0;
		TEMP_OFFSET :	REAL := 10.0;
		TEMP_HYS :	REAL := 5.0;
		T_MAX_HEAT :	TIME := t#10m;
		T_MAX_RET :	TIME := t#10m;
		TP_0 :	TIME := t#5m;
		TP_1 :	TIME := t#5m;
		TP_2 :	TIME := t#5m;
		TP_3 :	TIME := t#5m;
		TP_4 :	TIME := t#5m;
		TP_5 :	TIME := t#5m;
		TP_6 :	TIME := t#5m;
		TP_7 :	TIME := t#5m;
	END_VAR

	VAR_OUTPUT
		HEAT :	BOOL;
		PUMP :	BOOL;
		VALVE0 :	BOOL;
		VALVE1 :	BOOL;
		VALVE2 :	BOOL;
		VALVE3 :	BOOL;
		VALVE4 :	BOOL;
		VALVE5 :	BOOL;
		VALVE6 :	BOOL;
		VALVE7 :	BOOL;
		RUN :	BOOL;
		_STATUS :	BYTE;
	END_VAR

	VAR
		X1 :	TIMER_1_Block;
		x2 :	SEQUENCE_8_Block;
		x3 :	HYST_1_Block;
		init :	BOOL;
	END_VAR

	IF NOT init THEN
		init := TRUE;
		X1.day := SHR(BYTE#128,day);
		X1.start := T_start;
		X3.low := Temp_offset + temp_set;
		X3.high := Temp_hys + X3.low;
		X2.wait0 := T_max_heat;
		X2.delay0 := TP_0;
		X2.delay1 := TP_1;
		X2.delay2 := TP_2;
		X2.delay3 := TP_3;
		X2.delay4 := TP_4;
		X2.delay5 := TP_5;
		X2.delay6 := TP_6;
		X2.delay7 := TP_7;
		X2.wait1 := T_max_ret;
		X2.wait2 := T_max_ret;
		X2.wait3 := T_max_ret;
		X2.wait4 := T_max_ret;
		X2.wait5 := T_max_ret;
		X2.wait6 := T_max_ret;
		X2.wait7 := T_max_ret;
		X2();
	END_IF;

	X1(DTi := DT_in);
	IF X1.Q OR MANUAL OR x2.run THEN
		X3(in := temp_boiler);
		X2.in0 := X3.Q OR x3.win;
		X2.in1 := temp_return >= temp_set;
		X2.in2 := x2.in1;
		X2.in3 := x2.in1;
		X2.in4 := x2.in1;
		X2.in5 := x2.in1;
		X2.in6 := x2.in1;
		X2.in7 := x2.in1;
		X2.rst := rst;
		X2(start := X1.Q OR MANUAL);
		run := x2.run;
		pump := x2.QX;
		Heat := NOT X3.Q AND x2.run;
		valve0 := X2.Q0;
		valve1 := X2.Q1;
		valve2 := X2.Q2;
		valve3 := X2.Q3;
		valve4 := X2.Q4;
		valve5 := X2.Q5;
		valve6 := X2.Q6;
		valve7 := X2.Q7;
		pump := X2.QX;
		_STATUS := X2.status;
	ELSE
		X2(start := FALSE);
		_STATUS := x2.status;
	END_IF;

END_FUNCTION_BLOCK

PROGRAM program0
	VAR
		MANUAL :	BOOL;
		TEMP_BOILER :	REAL;
		TEMP_RETURN :	REAL := 100.0;
		DT_IN :	UDINT;
		RST :	BOOL;
		T_START :	UDINT := UDINT#10800000;(*tod#03:00:00*)
		DAY :	INT := 7;
		TEMP_SET :	REAL := 70.0;
		TEMP_OFFSET :	REAL := 10.0;
		TEMP_HYS :	REAL := 5.0;
		T_MAX_HEAT :	TIME := t#10m;
		T_MAX_RET :	TIME := t#10m;
		TP_0 :	TIME := t#5m;
		TP_1 :	TIME := t#5m;
		TP_2 :	TIME := t#5m;
		TP_3 :	TIME := t#5m;
		TP_4 :	TIME := t#5m;
		TP_5 :	TIME := t#5m;
		TP_6 :	TIME := t#5m;
		TP_7 :	TIME := t#5m;
		HEAT :	BOOL;
		PUMP :	BOOL;
		VALVE0 :	BOOL;
		VALVE1 :	BOOL;
		VALVE2 :	BOOL;
		VALVE3 :	BOOL;
		VALVE4 :	BOOL;
		VALVE5 :	BOOL;
		VALVE6 :	BOOL;
		VALVE7 :	BOOL;
		RUN :	BOOL;
		_STATUS :	BYTE;

		func_block : LEGIONELLA_Block;
	END_VAR
	func_block.MANUAL := MANUAL;
	func_block.TEMP_BOILER := TEMP_BOILER;
	func_block.TEMP_RETURN := TEMP_RETURN ;
	func_block.DT_IN    := DT_IN    ;
	func_block.RST := RST;
	func_block.T_START := T_START;
	func_block.DAY := DAY ;
	func_block.TEMP_SET := TEMP_SET ;
	func_block.TEMP_OFFSET    := TEMP_OFFSET    ;
	func_block.TEMP_HYS    := TEMP_HYS    ;
	func_block.T_MAX_HEAT := T_MAX_HEAT;
	func_block.T_MAX_RET := T_MAX_RET;
	func_block.TP_0 := TP_0;
	func_block.TP_1 := TP_1 ;
	func_block.TP_2 := TP_2 ;
	func_block.TP_3    := TP_3    ;
	func_block.TP_4    := TP_4    ;
	func_block.TP_5 := TP_5;
	func_block.TP_6 := TP_6;
	func_block.TP_7 := TP_7;

	func_block();
	HEAT  := func_block.HEAT;
	PUMP  := func_block.PUMP;
	VALVE0  := func_block.VALVE0;
	VALVE1  := func_block.VALVE1;
	VALVE2  := func_block.VALVE2;
	VALVE3  := func_block.HEAT;
	VALVE4  := func_block.VALVE4;
	VALVE5  := func_block.VALVE5;
	VALVE6  := func_block.VALVE6;
	VALVE7  := func_block.VALVE7;
	RUN  := func_block.RUN;
	_status  := func_block._status;
END_PROGRAM

CONFIGURATION Config0
	VAR_GLOBAL
		PLC_TICKS_PER_SEC :	INT;
		PLC_SYS_TICK_CNT :	DINT;
	END_VAR
  	RESOURCE Res0 ON PLC
    	TASK task0(INTERVAL := T#20ms,PRIORITY := 0);
    	PROGRAM instance0 WITH task0 : program0;
  	END_RESOURCE
END_CONFIGURATION

(* ---- LENGTH.ST ---- *)
FUNCTION_BLOCK LENGTH_Block

	VAR_INPUT
		M :	REAL;
		P :	REAL;
		IN :	REAL;
		FT :	REAL;
		YD :	REAL;
		MILE :	REAL;
		SM :	REAL;
		FM :	REAL;
	END_VAR

	VAR_OUTPUT
		YM :	REAL;
		YP :	REAL;
		YIN :	REAL;
		YFT :	REAL;
		YYD :	REAL;
		YMILE :	REAL;
		YSM :	REAL;
		YFM :	REAL;
	END_VAR

	Ym :=	m
			+ p * 0.000376065
			+ in * 0.0254
			+ ft * 0.3048
			+ yd * 0.9144
			+ mile * 1609.344
			+ sm * 1852.0
			+ fm * 1.829;
	Yp := Ym * 2659.11478068951;
	Yin := Ym * 39.37007874016;
	Yft := Ym * 3.28083989501;
	Yyd := Ym * 1.09361329834;
	Ymile := Ym * 0.00062137119;
	Ysm := Ym * 0.00053995680;
	Yfm := Ym * 0.54674685621;

END_FUNCTION_BLOCK

PROGRAM program0

	VAR
		M :	REAL;
		P :	REAL;
		IN :	REAL;
		FT :	REAL;
		YD :	REAL;
		MILE :	REAL;
		SM :	REAL;
		FM :	REAL;

		YM :	REAL;
		YP :	REAL;
		YIN :	REAL;
		YFT :	REAL;
		YYD :	REAL;
		YMILE :	REAL;
		YSM :	REAL;
		YFM :	REAL;

		func_block : LENGTH_Block;
	END_VAR
	func_block.M := M;
	func_block.P := P;
	func_block.IN := IN;
	func_block.FT := FT;
	func_block.YD := YD;
	func_block.MILE := MILE;
	func_block.SM := SM;
	func_block.FM := FM;

	func_block();

	YM := func_block.YM;
	YP := func_block.YP;
	YIN := func_block.YIN;
	YFT := func_block.YFT;
	YYD := func_block.YYD;
	YMILE := func_block.YMILE;
	YSM := func_block.YSM;
	YFM := func_block.YFM;

END_PROGRAM

CONFIGURATION Config0

	RESOURCE Res0 ON PLC
		TASK task0(INTERVAL := T#20ms,PRIORITY := 0);
		PROGRAM instance0 WITH task0 : program0;
	END_RESOURCE

END_CONFIGURATION

(* ---- LINEAR_INT.ST ---- *)
TYPE
	oscat_ARRAY_X               : ARRAY [0..1]    OF REAL;
	oscat_XY                    : ARRAY [1..20]   OF oscat_ARRAY_X := [0,0,0,0,0,0,0,0,0,0,0,0,0,0,0,0,0,0,0,0];
END_TYPE

FUNCTION_BLOCK LINEAR_INT_Block

	VAR_INPUT
		X :	REAL;
		XY :	oscat_XY;
		PTS :	INT;
	END_VAR

	VAR_OUTPUT
		LINEAR_INT :	REAL;
	END_VAR

	VAR
		i :	INT;
		i2 :	INT;
	END_VAR

	pts := MIN(pts,20);

	i := 2;

	WHILE (i < pts) AND (XY[i][0] < X) DO
		i := i + 1;
	END_WHILE;

	i2 := i-1;

	LINEAR_INT := ((XY[i][1] - XY[i2][1]) * X - XY[i][1] * XY[i2][0] + XY[i2][1] * XY[i][0]) / (XY[i][0] - XY[i2][0]);

END_FUNCTION_BLOCK

PROGRAM program0

	VAR
		X :	REAL;
		XY :	oscat_XY;
		PTS :	INT;

		LINEAR_INT :	REAL;

		func_block : LINEAR_INT_Block;
	END_VAR
	func_block.X := X;
	func_block.XY := XY;
	func_block.PTS := PTS;

	func_block();
	LINEAR_INT := func_block.LINEAR_INT;

END_PROGRAM

CONFIGURATION Config0

	RESOURCE Res0 ON PLC
		TASK task0(INTERVAL := T#20ms,PRIORITY := 0);
		PROGRAM instance0 WITH task0 : program0;
	END_RESOURCE

END_CONFIGURATION

(* ---- LIST_ADD.ST ---- *)
FUNCTION_BLOCK CHR_TO_STRING_Block
	VAR_INPUT
		C :	BYTE;
	END_VAR

	VAR_OUTPUT
		CHR_TO_STRING :	STRING;
	END_VAR

	CHR_TO_STRING := BYTE_TO_STRING(C);

END_FUNCTION_BLOCK

FUNCTION_BLOCK LIST_ADD_Block

	VAR_INPUT
		SEP :	BYTE;
		INS :	STRING;
	END_VAR

	VAR_IN_OUT
		LIST :	STRING;
	END_VAR

	VAR_OUTPUT
		LIST_ADD :	BOOL;
	END_VAR

	VAR
		CHR_TO_STRING :	CHR_TO_STRING_Block;
	END_VAR

	IF LEN(LIST) + LEN(INS) + 1 <= 250 THEN
	CHR_TO_STRING(C:=SEP);
	LIST := CONCAT(LIST, CHR_TO_STRING.CHR_TO_STRING);
	LIST := CONCAT(LIST, INS);
	LIST_ADD := TRUE;
	ELSE
	LIST_ADD := FALSE;
	END_IF;

END_FUNCTION_BLOCK

PROGRAM program0

	VAR
		SEP :	BYTE;
		INS :	STRING;

		LIST :	STRING;

		LIST_ADD :	BOOL;

		func_block : LIST_ADD_Block;
	END_VAR
	func_block.SEP := SEP;
	func_block.INS := INS;
	func_block.LIST := LIST;

	func_block();
	LIST := func_block.LIST;
	LIST_ADD := func_block.LIST_ADD;

END_PROGRAM

CONFIGURATION Config0

	RESOURCE Res0 ON PLC
		TASK task0(INTERVAL := T#20ms,PRIORITY := 0);
		PROGRAM instance0 WITH task0 : program0;
	END_RESOURCE

END_CONFIGURATION

(* ---- LOG_VIEWPORT.ST ---- *)
TYPE
  oscat_STRING80             : STRING;
  oscat_STRING250             : STRING;
END_TYPE

TYPE
  PRINTF_DATA_250  	:  ARRAY [1..11]  OF oscat_STRING250;
  PRINTF_DATA_80 	:  ARRAY [1..11]  OF oscat_STRING80;
  LOG_250       	:  ARRAY [0..400] OF oscat_STRING250;
  LOG_80    		:  ARRAY [0..400] OF oscat_STRING80;
  LOG_OPTION		:  ARRAY [0..400] OF DWORD;

  us_LOG_CONTROL :
  STRUCT
    NEW_MSG              : oscat_STRING250;    (*W neue Nachricht f�r den Datenbuffer   *)
	NEW_MSG_OPTION 		 : DWORD;
    LEVEL                : BYTE;
	SIZE                 : INT;                (*R Anzahl der Strings im LOG_DATA       *)
	RESET                : BOOL;               (*W Nachrichtenbuffer l�schen            *)
    PRINTF               : PRINTF_DATA_250;    (*W Array PRINTF Parameter               *)
    MSG                  : LOG_250;            (*I Array Message                        *)
    MSG_OPTION           : LOG_OPTION;     	   (*I Array Message Option                 *)
	UPDATE_COUNT         : UINT;               (*R Updatez�hler                         *)
    IDX                  : INT;                (*R aktueller Nachrichten-Index          *)
	RING_MODE            : BOOL;               (*I Buffer�berlauf erkannt               *)
  END_STRUCT;

  us_LOG_CONTROL_80 :
  STRUCT
    NEW_MSG              : oscat_STRING80;     (*W neue Nachricht f�r den Datenbuffer   *)
	NEW_MSG_OPTION 		 : DWORD;
    LEVEL                : BYTE;
	SIZE                 : INT;                (*R Anzahl der Strings im LOG_DATA       *)
	RESET                : BOOL;               (*W Nachrichtenbuffer l�schen            *)
    PRINTF               : PRINTF_DATA_80;     (*W Array PRINTF Parameter               *)
    MSG                  : LOG_80;             (*I Array Message                        *)
    MSG_OPTION           : LOG_OPTION;     	   (*I Array Message Option                 *)
	UPDATE_COUNT         : UINT;               (*R Updatez�hler                         *)
    IDX                  : INT;                (*R aktueller Nachrichten-Index          *)
	RING_MODE            : BOOL;               (*I Buffer�berlauf erkannt               *)
  END_STRUCT;

  LINE_ARRAY 			: ARRAY [1..40] OF INT;

  us_LOG_VIEWPORT :
    STRUCT
     LINE_ARRAY          : LINE_ARRAY;
     COUNT               : INT;                (* Anzahl der sichtbaren Nachtrichten   *)
	 UPDATE_COUNT        : UINT;               (* Updatez�hler                         *)
     MOVE_TO_X           : INT;                (* Steuerung der Nachrichtenanzeige     *)
     UPDATE              : BOOL;               (* Daten wurden ge�ndert -> neuzeichnen *)
  END_STRUCT;

END_TYPE

FUNCTION_BLOCK LOG_VIEWPORT_Block

  VAR_IN_OUT
    LC :	us_LOG_CONTROL_80;
    LV :	us_LOG_VIEWPORT;
  END_VAR

  VAR
    pos :	INT;
    count :	INT;
    idx :	INT;
    base :	INT;
    update_pos :	BOOL;
  END_VAR

  IF LV.MOVE_TO_X <> 0 THEN
    CASE LV.MOVE_TO_X OF
    30000:
      pos := 1 ;
    30001:
      pos := LC.SIZE;
    30002:
      pos := pos + LV.COUNT;
    30003:
      pos := pos - LV.COUNT;
    ELSE
      pos := pos + LV.MOVE_TO_X;
    END_CASE;
    update_pos := TRUE;
    LV.MOVE_TO_X := 0;
  END_IF;

  IF (LV.UPDATE_COUNT <> LC.UPDATE_COUNT) OR update_pos THEN
    LV.UPDATE := TRUE;
    LV.UPDATE_COUNT := LC.UPDATE_COUNT;
    update_pos := FALSE;

    IF LC.RING_MODE THEN
      pos := LIMIT(1,pos,LC.SIZE - LV.COUNT + 1);
    ELSE
      IF LC.IDX > LV.COUNT THEN
        pos := LIMIT(1,pos,LC.IDX - LV.COUNT + 1);
      ELSE
        pos := 1;
      END_IF;
    END_IF;

    base := LC.IDX - pos - LV.COUNT + 1;
    IF LC.RING_MODE THEN
      FOR count:= 1 TO LV.COUNT DO
        idx := base + count;
        IF idx < 1 THEN
          idx := idx + LC.SIZE;
        END_IF;
      END_FOR;
    ELSE
      FOR count:= 1 TO LV.COUNT DO
        idx := base + count;
        IF idx < 1 THEN
          LV.LINE_ARRAY[count] := 0;
        ELSE
          LV.LINE_ARRAY[count] := idx;
        END_IF;
      END_FOR;
    END_IF;
  END_IF;

END_FUNCTION_BLOCK

PROGRAM program0
	VAR
		LC :	us_LOG_CONTROL_80;
    LV :	us_LOG_VIEWPORT;

		func_block : LOG_VIEWPORT_Block;
	END_VAR
	func_block.LC := LC;
	func_block.LV := LV;

	func_block();
  LC  := func_block.LC;
  LV  := func_block.LV;

END_PROGRAM

CONFIGURATION Config0

  	RESOURCE Res0 ON PLC
    	TASK task0(INTERVAL := T#20ms,PRIORITY := 0);
    	PROGRAM instance0 WITH task0 : program0;
  	END_RESOURCE

END_CONFIGURATION

(* ---- LTCH.ST ---- *)
FUNCTION_BLOCK LTCH_Block

	VAR_INPUT
		D :	BOOL;
		L :	BOOL;
		RST :	BOOL;
	END_VAR

	VAR_OUTPUT
		Q :	BOOL;
	END_VAR

	IF rst THEN				(* if asynchronous reset then Q=0 *)
		Q := FALSE;
	ELSIF L THEN			(* latch is transparent *)
		Q := D;
	END_IF;

END_FUNCTION_BLOCK

PROGRAM program0

	VAR
		D :	BOOL;
		L :	BOOL;
		RST :	BOOL;

		Q :	BOOL;

		func_block : LTCH_Block;
	END_VAR
	func_block.D := D;
	func_block.L := L;
	func_block.RST := RST;

	func_block();
	Q := func_block.Q;

END_PROGRAM

CONFIGURATION Config0

	RESOURCE Res0 ON PLC
		TASK task0(INTERVAL := T#20ms,PRIORITY := 0);
		PROGRAM instance0 WITH task0 : program0;
	END_RESOURCE

END_CONFIGURATION

(* ---- LTCH_4.ST ---- *)
FUNCTION_BLOCK LTCH_4_Block

	VAR_INPUT
		D0 :	BOOL;
		D1 :	BOOL;
		D2 :	BOOL;
		D3 :	BOOL;
		L :	BOOL;
		RST :	BOOL;
	END_VAR

	VAR_OUTPUT
		Q0 :	BOOL;
		Q1 :	BOOL;
		Q2 :	BOOL;
		Q3 :	BOOL;
	END_VAR

	IF rst THEN			(* if asynchronous reset then Q=0 *)
		Q0 := FALSE;
		Q1 := FALSE;
		Q2 := FALSE;
		Q3 := FALSE;
	ELSIF L THEN			(* latch is transparent *)
		Q0 := D0;
		Q1 := D1;
		Q2 := D2;
		Q3 := D3;
	END_IF;

END_FUNCTION_BLOCK

PROGRAM program0

	VAR
		D0 :	BOOL;
		D1 :	BOOL;
		D2 :	BOOL;
		D3 :	BOOL;
		L :	BOOL;
		RST :	BOOL;

		Q0 :	BOOL;
		Q1 :	BOOL;
		Q2 :	BOOL;
		Q3 :	BOOL;

		func_block : LTCH_4_Block;
	END_VAR
	func_block.D0 := D0;
	func_block.D1 := D1;
	func_block.D2 := D2;
	func_block.D3 := D3;
	func_block.L := L;
	func_block.RST := RST;

	func_block();
	Q0 := func_block.Q0;
	Q1 := func_block.Q1;
	Q2 := func_block.Q2;
	Q3 := func_block.Q3;

END_PROGRAM

CONFIGURATION Config0

	RESOURCE Res0 ON PLC
		TASK task0(INTERVAL := T#20ms,PRIORITY := 0);
		PROGRAM instance0 WITH task0 : program0;
	END_RESOURCE

END_CONFIGURATION

(* ---- M_D.ST ---- *)
FUNCTION_BLOCK T_PLC_MS_Block
	VAR_OUTPUT
		T_PLC_MS :	UDINT;
	END_VAR

	VAR_EXTERNAL
		PLC_TICKS_PER_SEC :	INT;
		PLC_SYS_TICK_CNT :	DINT;
	END_VAR

	VAR
		debug :	BOOL;(*Debug-Mode ON / OFF*)
		N :	INT;(*Debug-Faktor*)
		Offset :	UDINT;(*Debug-Offset*)
		temp :	DWORD := DWORD#1;(*Debug-Offset*)
		mode :	BOOL;(*modus*)
		faktor :	UDINT;(*Systemtakt-Faktor*)
		init :	BOOL;
		v_plc_ticks_per_sec :	UDINT;
		base :	UDINT := UDINT#1000;
	END_VAR

	IF init = FALSE THEN
		v_plc_ticks_per_sec := INT_TO_UDINT(PLC_TICKS_PER_SEC);
		IF v_plc_ticks_per_sec = UDINT#1024 THEN
			faktor := UDINT#1;
			mode := FALSE;
		ELSIF v_plc_ticks_per_sec > UDINT#0 THEN
			IF v_plc_ticks_per_sec <= base THEN
				faktor := base / v_plc_ticks_per_sec;
				mode := FALSE;
			ELSE
				faktor := v_plc_ticks_per_sec / base;
				mode := TRUE;
			END_IF;
		ELSE
			faktor := UDINT#1;
		END_IF;
		init := TRUE;
	END_IF;

	IF mode THEN
		T_PLC_MS := DINT_TO_UDINT(PLC_SYS_TICK_CNT) / faktor;
	ELSE
		T_PLC_MS := DINT_TO_UDINT(PLC_SYS_TICK_CNT) * faktor;
	END_IF;

	IF debug THEN
		T_PLC_MS := (DWORD_TO_UDINT(SHL(UDINT_TO_DWORD(T_PLC_MS),N) OR SHL(temp,N)) - UDINT#1) + Offset;
	END_IF;
END_FUNCTION_BLOCK

FUNCTION_BLOCK M_D_Block

	VAR_INPUT
		START :	BOOL;
		STOP :	BOOL;
		TMAX :	TIME := t#10d;
		RST :	BOOL;
	END_VAR

	VAR_OUTPUT
		PT :	TIME;
		ET :	TIME;
		RUN :	BOOL;
	END_VAR

	VAR
		edge :	BOOL;
		T0 :	TIME;
		tx :	TIME;
		startup :	BOOL;
		T_PLC_MS :	T_PLC_MS_Block;
	END_VAR

	(* check for rst input *)
	IF rst OR et >= tmax THEN
		pt := t#0ms;
		et := t#0ms;
		startup := FALSE;
		run := FALSE;
	END_IF;

	(* avoid timers to start when input is true at startup *)
	IF NOT startup THEN
		edge := start;
		startup := TRUE;
	END_IF;

	(* read system timer *)
	T_PLC_MS();
	tx:= UDINT_TO_TIME(T_PLC_MS.T_PLC_MS);

	(* detect rising edge on start *)
	IF start AND NOT edge AND NOT stop THEN
		t0 := tx;
		run := TRUE;
		pt := t#0s;
	ELSIF stop AND run THEN
		pt := et;
		run := FALSE;
	END_IF;
	edge := start;
	IF run THEN et := tx - t0; END_IF;

END_FUNCTION_BLOCK

PROGRAM program0

	VAR
		START :	BOOL;
		STOP :	BOOL;
		TMAX :	TIME := t#10d;
		RST :	BOOL;

		PT :	TIME;
		ET :	TIME;
		RUN :	BOOL;

		func_block : M_D_Block;
	END_VAR
	func_block.START := START;
	func_block.STOP := STOP;
	func_block.TMAX := TMAX;
	func_block.RST := RST;

	func_block();
	PT := func_block.PT;
	ET := func_block.ET;
	RUN := func_block.RUN;

END_PROGRAM

CONFIGURATION Config0

	VAR_GLOBAL
		PLC_TICKS_PER_SEC :	INT;
		PLC_SYS_TICK_CNT :	DINT;
	END_VAR

	RESOURCE Res0 ON PLC
		TASK task0(INTERVAL := T#20ms,PRIORITY := 0);
		PROGRAM instance0 WITH task0 : program0;
	END_RESOURCE

END_CONFIGURATION

(* ---- M_T.ST ---- *)
FUNCTION_BLOCK T_PLC_MS_block
	VAR_OUTPUT
		T_PLC_MS :	UDINT;
	END_VAR

	VAR_EXTERNAL
		PLC_TICKS_PER_SEC :	INT;
		PLC_SYS_TICK_CNT :	DINT;
	END_VAR

	VAR
		debug :	BOOL;(*Debug-Mode ON / OFF*)
		N :	INT;(*Debug-Faktor*)
		Offset :	UDINT;(*Debug-Offset*)
		temp :	DWORD := DWORD#1;(*Debug-Offset*)
		mode :	BOOL;(*modus*)
		faktor :	UDINT;(*Systemtakt-Faktor*)
		init :	BOOL;
		v_plc_ticks_per_sec :	UDINT;
		base :	UDINT := UDINT#1000;
	END_VAR

	IF init = FALSE THEN
		v_plc_ticks_per_sec := INT_TO_UDINT(PLC_TICKS_PER_SEC);
		IF v_plc_ticks_per_sec = UDINT#1024 THEN
			faktor := UDINT#1;
			mode := FALSE;
		ELSIF v_plc_ticks_per_sec > UDINT#0 THEN
			IF v_plc_ticks_per_sec <= base THEN
				faktor := base / v_plc_ticks_per_sec;
				mode := FALSE;
			ELSE
				faktor := v_plc_ticks_per_sec / base;
				mode := TRUE;
			END_IF;
		ELSE
			faktor := UDINT#1;
		END_IF;
		init := TRUE;
	END_IF;

	IF mode THEN
		T_PLC_MS := DINT_TO_UDINT(PLC_SYS_TICK_CNT) / faktor;
	ELSE
		T_PLC_MS := DINT_TO_UDINT(PLC_SYS_TICK_CNT) * faktor;
	END_IF;

	IF debug THEN
		T_PLC_MS := (DWORD_TO_UDINT(SHL(UDINT_TO_DWORD(T_PLC_MS),N) OR SHL(temp,N)) - UDINT#1) + Offset;
	END_IF;
END_FUNCTION_BLOCK

FUNCTION_BLOCK M_T_Block

	VAR_INPUT
		IN :	BOOL;
		TMAX :	TIME := t#10d;
		RST :	BOOL;
	END_VAR

	VAR_OUTPUT
		PT :	TIME;
		ET :	TIME;
	END_VAR

	VAR
		edge :	BOOL;
		start :	TIME;
		tx :	TIME;
		T_PLC_MS :	T_PLC_MS_Block;
	END_VAR

	(*@KEY@: WORKSHEET
	NAME: M_T
	IEC_LANGUAGE: ST
	*)
	(* read system timer *)
	T_PLC_MS();
	tx:= UDINT_TO_TIME(T_PLC_MS.T_PLC_MS);

	IF RST OR ET >= TMAX THEN
		PT := t#0s;
		ET := PT;
	ELSIF IN THEN
		IF NOT edge THEN start := tx; END_IF;
		ET := tx - start;
	ELSE
		PT := ET;
	END_IF;
	edge := IN;

END_FUNCTION_BLOCK

PROGRAM program0

	VAR
		IN :	BOOL;
		TMAX :	TIME := t#10d;
		RST :	BOOL;

		PT :	TIME;
		ET :	TIME;

		func_block : M_T_Block;
	END_VAR
	func_block.IN := IN;
	func_block.TMAX := TMAX;
	func_block.RST := RST;

	func_block();
	PT := func_block.PT;
	ET := func_block.ET;

END_PROGRAM

CONFIGURATION Config0

	VAR_GLOBAL
		PLC_TICKS_PER_SEC :	INT;
		PLC_SYS_TICK_CNT :	DINT;
	END_VAR

	RESOURCE Res0 ON PLC
		TASK task0(INTERVAL := T#20ms,PRIORITY := 0);
		PROGRAM instance0 WITH task0 : program0;
	END_RESOURCE

END_CONFIGURATION

(* ---- M_TX.ST ---- *)
FUNCTION_BLOCK T_PLC_MS_block
	VAR_OUTPUT
		T_PLC_MS :	UDINT;
	END_VAR

	VAR_EXTERNAL
		PLC_TICKS_PER_SEC :	INT;
		PLC_SYS_TICK_CNT :	DINT;
	END_VAR

	VAR
		debug :	BOOL;(*Debug-Mode ON / OFF*)
		N :	INT;(*Debug-Faktor*)
		Offset :	UDINT;(*Debug-Offset*)
		temp :	DWORD := DWORD#1;(*Debug-Offset*)
		mode :	BOOL;(*modus*)
		faktor :	UDINT;(*Systemtakt-Faktor*)
		init :	BOOL;
		v_plc_ticks_per_sec :	UDINT;
		base :	UDINT := UDINT#1000;
	END_VAR

	IF init = FALSE THEN
		v_plc_ticks_per_sec := INT_TO_UDINT(PLC_TICKS_PER_SEC);
		IF v_plc_ticks_per_sec = UDINT#1024 THEN
			faktor := UDINT#1;
			mode := FALSE;
		ELSIF v_plc_ticks_per_sec > UDINT#0 THEN
			IF v_plc_ticks_per_sec <= base THEN
				faktor := base / v_plc_ticks_per_sec;
				mode := FALSE;
			ELSE
				faktor := v_plc_ticks_per_sec / base;
				mode := TRUE;
			END_IF;
		ELSE
			faktor := UDINT#1;
		END_IF;
		init := TRUE;
	END_IF;

	IF mode THEN
		T_PLC_MS := DINT_TO_UDINT(PLC_SYS_TICK_CNT) / faktor;
	ELSE
		T_PLC_MS := DINT_TO_UDINT(PLC_SYS_TICK_CNT) * faktor;
	END_IF;

	IF debug THEN
		T_PLC_MS := (DWORD_TO_UDINT(SHL(UDINT_TO_DWORD(T_PLC_MS),N) OR SHL(temp,N)) - UDINT#1) + Offset;
	END_IF;
END_FUNCTION_BLOCK

FUNCTION_BLOCK M_TX_Block

	VAR_INPUT
		IN :	BOOL;
		TMAX :	TIME := t#10d;
		RST :	BOOL;
	END_VAR

	VAR_OUTPUT
		TH :	TIME;
		TL :	TIME;
		DC :	REAL;
		F :	REAL;
		ET :	TIME;
	END_VAR

	VAR
		edge :	BOOL;
		start :	TIME;
		stop :	TIME;
		tx :	TIME;
		rise :	BOOL;
		fall :	BOOL;
		startup :	BOOL;
		T_PLC_MS :	T_PLC_MS_block;
	END_VAR

	IF rst OR (et >= tmax) THEN
		rise := FALSE;
		fall := FALSE;
		startup := FALSE;
		th := t#0ms;
		tl := t#0ms;
		DC := 0.0;
		F := 0.0;
		ET := t#0s;
	END_IF;

	(* avoid timers to start when input is true at startup *)
	IF NOT startup THEN
		edge := in;
		startup := TRUE;
	END_IF;

	(* read system timer *)
	T_PLC_MS();
	tx:= UDINT_TO_TIME(T_PLC_MS.T_PLC_MS);

	(* edge trigger rising and falling edge *)
	IF in XOR edge THEN
		edge := in;
		(* rising edge starts measurement *)
		IF in THEN
			start := Tx;
			rise := TRUE;
			IF fall THEN tl := start - stop; END_IF;
			IF th > t#0ms AND tl > t#0ms THEN
				dc := TIME_TO_REAL(th) / TIME_TO_REAL(th+tl);
				f := 1000.0 / TIME_TO_REAL(th + tl);
			END_IF;
		(* falling edge starts second cycle measurement *)
		ELSE
			stop := Tx;
			fall := TRUE;
			IF rise THEN th := stop - start; END_IF;
			IF th > t#0ms AND tl > t#0ms THEN
				dc := TIME_TO_REAL(th) /  TIME_TO_REAL(th+tl);
				f := 1000.0 / TIME_TO_REAL(th + tl);
			END_IF;
		END_IF;
	END_IF;
	IF rise THEN et := tx - start; END_IF;

	(* check FOR rst input *)
	IF rst OR (et >= tmax) THEN
		rise := FALSE;
		fall := FALSE;
		startup := FALSE;
		th := t#0ms;
		tl := t#0ms;
		DC := 0.0;
		F := 0.0;
		ET := t#0s;
	END_IF;

	(* avoid timers to start when input is true at startup *)
	IF NOT startup THEN
		edge := in;
		startup := TRUE;
	END_IF;

	(* read system timer *)
	T_PLC_MS();
	tx:= UDINT_TO_TIME(T_PLC_MS.T_PLC_MS);

	(* edge trigger rising and falling edge *)
	IF in XOR edge THEN
		edge := in;
		(* rising edge starts measurement *)
		IF in THEN
			start := Tx;
			rise := TRUE;
			IF fall THEN tl := start - stop; END_IF;
			IF th > t#0ms AND tl > t#0ms THEN
				dc := TIME_TO_REAL(th) / TIME_TO_REAL(th+tl);
				f := 1000.0 / TIME_TO_REAL(th + tl);
			END_IF;
		(* falling edge starts second cycle measurement *)
		ELSE
			stop := Tx;
			fall := TRUE;
			IF rise THEN th := stop - start; END_IF;
			IF th > t#0ms AND tl > t#0ms THEN
				dc := TIME_TO_REAL(th) /  TIME_TO_REAL(th+tl);
				f := 1000.0 / TIME_TO_REAL(th + tl);
			END_IF;
		END_IF;
	END_IF;
	IF rise THEN et := tx - start; END_IF;

END_FUNCTION_BLOCK

PROGRAM program0

	VAR
		IN :	BOOL;
		TMAX :	TIME := t#10d;
		RST :	BOOL;

		TH :	TIME;
		TL :	TIME;
		DC :	REAL;
		F :	REAL;
		ET :	TIME;

		func_block : M_TX_Block;
	END_VAR
	func_block.IN := IN;
	func_block.TMAX := TMAX;
	func_block.RST := RST;

	func_block();
	TH := func_block.TH;
	TL := func_block.TL;
	DC := func_block.DC;
	F := func_block.F;
	ET := func_block.ET;

END_PROGRAM

CONFIGURATION Config0

	VAR_GLOBAL
		PLC_TICKS_PER_SEC :	INT;
		PLC_SYS_TICK_CNT :	DINT;
	END_VAR

	RESOURCE Res0 ON PLC
		TASK task0(INTERVAL := T#20ms,PRIORITY := 0);
		PROGRAM instance0 WITH task0 : program0;
	END_RESOURCE

END_CONFIGURATION

(* ---- MANUAL_1.ST ---- *)
FUNCTION_BLOCK MANUAL_1_Block

	VAR_INPUT
		_IN :	BOOL;
		MAN :	BOOL;
		M_I :	BOOL;
		SET :	BOOL;
		RST :	BOOL;
	END_VAR

	VAR_OUTPUT
		Q :	BOOL;
		STATUS :	BYTE;
	END_VAR

	VAR
		S_edge :	BOOL;
		_r_edge :	BOOL;
		edge :	BOOL;
	END_VAR

	IF NOT man THEN
		Q := _IN;
		STATUS := BYTE#100;
		edge := FALSE;
	ELSIF NOT s_edge AND set THEN
		Q := TRUE;
		edge := TRUE;
		status := BYTE#101;
	ELSIF NOT _r_edge AND rst THEN
		Q := FALSE;
		edge := TRUE;
		status := BYTE#102;
	ELSIF NOT edge THEN
		Q := M_I;
		status := BYTE#103;
	END_IF;

	(* remember levels of manual signals *)
	s_edge := SET;
	_r_edge := RST;

END_FUNCTION_BLOCK

PROGRAM program0

	VAR
		_IN :	BOOL;
		MAN :	BOOL;
		M_I :	BOOL;
		SET :	BOOL;
		RST :	BOOL;

		Q :	BOOL;
		STATUS :	BYTE;

		func_block : MANUAL_1_Block;
	END_VAR
	func_block._IN := _IN;
	func_block.MAN := MAN;
	func_block.M_I := M_I;
	func_block.SET := SET;
	func_block.RST := RST;
	func_block();
	Q := func_block.Q;
	STATUS := func_block.STATUS;

END_PROGRAM

CONFIGURATION Config0

	RESOURCE Res0 ON PLC
		TASK task0(INTERVAL := T#20ms,PRIORITY := 0);
		PROGRAM instance0 WITH task0 : program0;
	END_RESOURCE

END_CONFIGURATION

(* ---- MANUAL_2.ST ---- *)
FUNCTION_BLOCK MANUAL_2_Block

	VAR_INPUT
		_IN :	BOOL;
		ENA :	BOOL;
		_ON :	BOOL;
		OFF :	BOOL;
		MAN :	BOOL;
	END_VAR

	VAR_OUTPUT
		Q :	BOOL;
		STATUS :	BYTE;
	END_VAR

	IF ena THEN
		IF NOT _ON AND NOT OFF THEN
			Q := _IN;
			STATUS := BYTE#100;
		ELSIF _on AND NOT off THEN
			Q := TRUE;
			STATUS := BYTE#101;
		ELSIF NOT _on AND off THEN
			q := FALSE;
			STATUS := BYTE#102;
		ELSE
			Q := MAN;
			STATUS := BYTE#103;
		END_IF;
	ELSE
		Q := FALSE;
		STATUS := BYTE#104;
	END_IF;

END_FUNCTION_BLOCK

PROGRAM program0

	VAR
		_IN :	BOOL;
		ENA :	BOOL;
		_ON :	BOOL;
		OFF :	BOOL;
		MAN :	BOOL;

		Q :	BOOL;
		STATUS :	BYTE;

		func_block : MANUAL_2_Block;
	END_VAR
	func_block._IN := _IN;
	func_block.ENA := ENA;
	func_block._ON := _ON;
	func_block.OFF := OFF;
	func_block.MAN := MAN;
	func_block();
	Q := func_block.Q;
	STATUS := func_block.STATUS;

END_PROGRAM

CONFIGURATION Config0

	RESOURCE Res0 ON PLC
		TASK task0(INTERVAL := T#20ms,PRIORITY := 0);
		PROGRAM instance0 WITH task0 : program0;
	END_RESOURCE

END_CONFIGURATION

(* ---- MANUAL_4.ST ---- *)
FUNCTION INC:INT
	VAR_INPUT
		X :	INT;
		D :	INT;
		M :	INT;
	END_VAR

	inc := (X + D + M + 1) MOD (M + 1);
END_FUNCTION

FUNCTION_BLOCK MANUAL_4_Block

	VAR_INPUT
		I0 :	BOOL;
		I1 :	BOOL;
		I2 :	BOOL;
		I3 :	BOOL;
		MAN :	BOOL;
		STP :	BOOL;
		M0 :	BOOL;
		M1 :	BOOL;
		M2 :	BOOL;
		M3 :	BOOL;
	END_VAR

	VAR_OUTPUT
		Q0 :	BOOL;
		Q1 :	BOOL;
		Q2 :	BOOL;
		Q3 :	BOOL;
		STATUS :	BYTE;
	END_VAR

	VAR
		edge :	BOOL;
		pos :	INT;
		tog :	BOOL;
	END_VAR

	IF man THEN
		IF NOT TOG THEN
			Q0 := M0;
			Q1 := M1;
			Q2 := M2;
			Q3 := M3;
			STATUS := BYTE#101;
		END_IF;
		IF STP AND NOT edge THEN
			tog := TRUE;
			CASE pos OF
				0:	Q0 := TRUE;
					Q1 := FALSE;
					Q2 := FALSE;
					Q3 := FALSE;
					STATUS := BYTE#110;
				1:	Q0 := FALSE;
					Q1 := TRUE;
					Q2 := FALSE;
					Q3 := FALSE;
					STATUS := BYTE#111;
				2:	Q0 := FALSE;
					Q1 := FALSE;
					Q2 := TRUE;
					Q3 := FALSE;
					STATUS := BYTE#112;
				3:	Q0 := FALSE;
					Q1 := FALSE;
					Q2 := FALSE;
					Q3 := TRUE;
					STATUS := BYTE#113;
			END_CASE;
			pos := INC(pos,1,3);
		END_IF;
	ELSE
		Q0 := I0;
		Q1 := I1;
		Q2 := I2;
		Q3 := I3;
		STATUS := BYTE#100;
		tog := FALSE;
		pos := 0;
	END_IF;

	edge := STP;

END_FUNCTION_BLOCK

PROGRAM program0

	VAR
		I0 :	BOOL;
		I1 :	BOOL;
		I2 :	BOOL;
		I3 :	BOOL;
		MAN :	BOOL;
		STP :	BOOL;
		M0 :	BOOL;
		M1 :	BOOL;
		M2 :	BOOL;
		M3 :	BOOL;

		Q0 :	BOOL;
		Q1 :	BOOL;
		Q2 :	BOOL;
		Q3 :	BOOL;
		STATUS :	BYTE;

		func_block : MANUAL_4_Block;
	END_VAR
	func_block.I0 := I0;
	func_block.I1 := I1;
	func_block.I2 := I2;
	func_block.I3 := I3;
	func_block.MAN := MAN;
	func_block.STP := STP;
	func_block.M0 := M0;
	func_block.M1 := M1;
	func_block.M2 := M2;
	func_block.M3 := M3;
	func_block();
	Q0 := func_block.Q0;
	Q1 := func_block.Q1;
	Q2 := func_block.Q2;
	Q3 := func_block.Q3;
	STATUS := func_block.STATUS;

END_PROGRAM

CONFIGURATION Config0

	RESOURCE Res0 ON PLC
		TASK task0(INTERVAL := T#20ms,PRIORITY := 0);
		PROGRAM instance0 WITH task0 : program0;
	END_RESOURCE

END_CONFIGURATION

(* ---- MATRIX.ST ---- *)
TYPE
	oscat_arb_0_3               : ARRAY [0..3]    OF BYTE;
END_TYPE

FUNCTION BIT_OF_DWORD : BOOL
	VAR_INPUT
		IN : DWORD;
		N : INT;
	END_VAR

	BIT_OF_DWORD := (SHR(in,N) AND 16#00000001) > 0;
END_FUNCTION

FUNCTION _BYTE_TO_INT:INT
	VAR_INPUT
		IN :	BYTE;
	END_VAR

	_BYTE_TO_INT := USINT_TO_INT(BYTE_TO_USINT(IN));
END_FUNCTION

FUNCTION BIT_LOAD_B:BYTE
	VAR_INPUT
		IN :	BYTE;
		VAL :	BOOL;
		POS :	INT;
	END_VAR

	IF VAL THEN
		BIT_LOAD_B := in OR SHL(BYTE#1,pos);
	ELSE
		BIT_LOAD_B := in AND (NOT SHL(BYTE#1,pos));
	END_IF;
END_FUNCTION

FUNCTION_BLOCK MATRIX_Block

	VAR_INPUT
		X1 :	BOOL;
		X2 :	BOOL;
		X3 :	BOOL;
		X4 :	BOOL;
		X5 :	BOOL;
		RELEASE :	BOOL;
	END_VAR

	VAR_OUTPUT
		CODE :	BYTE;
		_TP :	BOOL;
		Y1 :	BOOL := TRUE;
		Y2 :	BOOL;
		Y3 :	BOOL;
		Y4 :	BOOL;
	END_VAR

	VAR
		line :	BYTE;
		X :	oscat_arb_0_3;
		L :	oscat_arb_0_3;
		i :	INT;
		temp :	BYTE;
		temp2 :	BYTE;
		L_temp :	BYTE;
		temp_bit :	BOOL;
		in_temp :	INT;
	END_VAR

	_TP := FALSE;
	code := BYTE#0;

	(* read scan lines *)
	in_temp := _BYTE_TO_INT(line);
	temp := X[in_temp];  (* X[LINE] umkopieren *)

	temp:=BIT_LOAD_B(temp,X1,0); (* X[line].0 := X1; *)
	temp:=BIT_LOAD_B(temp,X2,1); (* X[line].1 := X2; *)
	temp:=BIT_LOAD_B(temp,X3,2); (* X[line].2 := X3; *)
	temp:=BIT_LOAD_B(temp,X4,3); (* X[line].3 := X4; *)
	temp:=BIT_LOAD_B(temp,X5,4); (* X[line].4 := X5; *)

	X[in_temp] := temp; (* X[LINE] zur�ckkopieren *)

	(* compare for change *)
	FOR i := 0 TO 3 DO
		IF X[i] <> L[i] THEN
			(* scan line information has changed code need to be found and generated *)
			temp   := x[i] XOR L[i];
			temp2  := X[i];
			L_temp := L[i];

			IF BIT_OF_DWORD(BYTE_TO_DWORD(temp),0) THEN (* temp.X0 *)
				code := BYTE#1;
				temp_bit := BIT_OF_DWORD(BYTE_TO_DWORD(temp2),0);   (* X[i].X0 *)
				code := BIT_LOAD_B(code,temp_bit,7);     			(* code.X7 *)
				L_temp := BIT_LOAD_B(L_temp,temp_bit,0); 			(* L[i].X0 *)
			ELSIF BIT_OF_DWORD(BYTE_TO_DWORD(temp),1) THEN          (* temp.X1 *)
				code := BYTE#2;
				temp_bit := BIT_OF_DWORD(BYTE_TO_DWORD(temp2),1);   (* X[i].X1 *)
				code := BIT_LOAD_B(code,temp_bit,7);     			(* code.X7 *)
				L_temp := BIT_LOAD_B(L_temp,temp_bit,1); 			(* L[i].X1 *)
			ELSIF BIT_OF_DWORD(BYTE_TO_DWORD(temp),2) THEN          (* temp.X2 *)
				code := BYTE#3;
				temp_bit := BIT_OF_DWORD(BYTE_TO_DWORD(temp2),2);   (* X[i].X2 *)
				code := BIT_LOAD_B(code,temp_bit,7);     			(* code.X7 *)
				L_temp := BIT_LOAD_B(L_temp,temp_bit,2); 			(* L[i].X2 *)
			ELSIF BIT_OF_DWORD(BYTE_TO_DWORD(temp),3) THEN          (* temp.X3 *)
				code := BYTE#4;
				temp_bit := BIT_OF_DWORD(BYTE_TO_DWORD(temp2),3);   (* X[i].X3 *)
				code := BIT_LOAD_B(code,temp_bit,7);     			(* code.X7 *)
				L_temp := BIT_LOAD_B(L_temp,temp_bit,3); 			(* L[i].X3 *)
			ELSIF BIT_OF_DWORD(BYTE_TO_DWORD(temp),4) THEN          (* temp.X4 *)
				code := BYTE#5;
				temp_bit := BIT_OF_DWORD(BYTE_TO_DWORD(temp2),4);   (* X[i].X4 *)
				code := BIT_LOAD_B(code,temp_bit,7);     			(* code.X7 *)
				L_temp := BIT_LOAD_B(L_temp,temp_bit,4); 			(* L[i].X4 *)
			END_IF;
			L[i] := L_temp;
			_TP := TRUE;
			code := (code AND BYTE#2#1000_1111) OR SHL(LINE AND BYTE#2#0000_0111,4);
			(* obere zeile enspricht: Code.X4 := Line.X0; /  Code.X5 := Line.X1; / Code.X6 := Line.X2; *)

			(* check if release codes need to be killed *)
			IF NOT release AND code < BYTE#127 THEN
				code := BYTE#0;
				_TP := FALSE;
			END_IF;
			EXIT;
		END_IF;
	END_FOR;

	(* increment scan line every cycle *)
	line := INT_TO_BYTE(_BYTE_TO_INT(line) + 1) AND BYTE#2#0000_0011;
	temp := SHL(BYTE#1,_BYTE_TO_INT(line));

	Y1 := BIT_OF_DWORD(BYTE_TO_DWORD(temp),0); (* temp.0 *)
	Y2 := BIT_OF_DWORD(BYTE_TO_DWORD(temp),1); (* temp.1 *)
	Y3 := BIT_OF_DWORD(BYTE_TO_DWORD(temp),2); (* temp.2 *)
	Y4 := BIT_OF_DWORD(BYTE_TO_DWORD(temp),3); (* temp.3 *)

END_FUNCTION_BLOCK

PROGRAM program0

	VAR
		X1 :	BOOL;
		X2 :	BOOL;
		X3 :	BOOL;
		X4 :	BOOL;
		X5 :	BOOL;
		RELEASE :	BOOL;

		CODE :	BYTE;
		_TP :	BOOL;
		Y1 :	BOOL := TRUE;
		Y2 :	BOOL;
		Y3 :	BOOL;
		Y4 :	BOOL;

		func_block : MATRIX_Block;
	END_VAR
	func_block.X1 := X1;
	func_block.X2 := X2;
	func_block.X3 := X3;
	func_block.X4 := X4;
	func_block.X5 := X5;
	func_block.RELEASE := RELEASE;
	func_block();
	CODE := func_block.CODE;
	_TP := func_block._TP;
	Y1 := func_block.Y1;
	Y2 := func_block.Y2;
	Y3 := func_block.Y3;
	Y4 := func_block.Y4;

END_PROGRAM

CONFIGURATION Config0

	RESOURCE Res0 ON PLC
		TASK task0(INTERVAL := T#20ms,PRIORITY := 0);
		PROGRAM instance0 WITH task0 : program0;
	END_RESOURCE

END_CONFIGURATION

(* ---- MB_CLIENT.ST ---- *)
TYPE
  oscat_IP_FIFO128_DATA  : ARRAY [1..128] OF BYTE;
  oscat_Mailbox  : ARRAY [1..16] OF BYTE;

  oscat_IP_FIFO_DATA :
  STRUCT
	X       : oscat_IP_FIFO128_DATA; (* IP_ID FIFO Speicher          *)
	Y       : oscat_IP_FIFO128_DATA; (* IP_ID Z�hler                 *)
	ID      : BYTE;                  (* h�chste vergabene id         *)
	MAX_ID  : BYTE;                  (* maximal Anmeldungen pro ID   *)
    INIT    : BOOL;                  (* Initialisierung durchgef�hrt *)
	EMPTY   : BOOL;                  (* FIFO leer                    *)
	FULL    : BOOL;                  (* FIFO voll                    *)
	TOP     : INT;                   (* maximale anzahl in FIFO      *)
	NW      : INT;                   (* Schreibzeiger                *)
	NR      : INT;                   (* Lesezeiger                   *)
  END_STRUCT;

  oscat_IP_C:
  STRUCT
  	C_MODE:			BYTE;          		(*W Mode: TCP/UCP AKTIV/PASSIV                               *)
	C_PORT:         WORD;          		(*W Portnummer                                               *)
	C_IP:           DWORD;         		(*W IP-Adresse gepackt wwxxyyzz = www.xxx.yyy.zzz            *)
    C_STATE:        BYTE;          		(*R Verbindungsstatus ON/OFF + Flanke ON/OFF                 *)
	C_ENABLE:       BOOL;          		(*W Freigabe f�r Connect                                     *)
    R_OBSERVE:      BOOL;          		(*W Empfang ueberwachen                                      *)
    TIME_RESET:     BOOL;          		(*W Alle Timer ruecksetzen                                   *)
	ERROR:          DWORD;         		(*R vvwwxxyy (vv = CON_ERROR, ww = SEN_ERROR, xx = REC_ERROR *)
    FIFO:           oscat_IP_FIFO_DATA; (*I IP FIFO Struktur                                         *)
	MAILBOX:		oscat_Mailbox;		(*I Mailbox: Datenbereich f�r Bausteindatenaustausch         *)
  END_STRUCT;
END_TYPE

TYPE
	oscat_aW0_255	: ARRAY [0..255] OF WORD;
	oscat_NW_BUF_SHORT : ARRAY [0..1407] OF BYTE;
	oscat_NW_BUF_LONG  : ARRAY [0..4095] OF BYTE;

	oscat_NETWORK_BUFFER_SHORT :
	STRUCT
		SIZE   : UINT;
		BUFFER : oscat_NW_BUF_SHORT;
	END_STRUCT;

	oscat_NETWORK_BUFFER :
	STRUCT
		SIZE   : UINT;
		BUFFER : oscat_NW_BUF_LONG;
	END_STRUCT;

END_TYPE

FUNCTION _BYTE_TO_INT:INT
	VAR_INPUT
		IN :	BYTE;
	END_VAR

	_BYTE_TO_INT := USINT_TO_INT(BYTE_TO_USINT(IN));
END_FUNCTION

FUNCTION_BLOCK IP_FIFO_Block

  VAR_IN_OUT
    FIFO :	oscat_IP_FIFO_DATA;
    ID :	BYTE;
    STATE :	BYTE;
  END_VAR

  VAR
    tmp :	INT;
  END_VAR

  IF NOT FIFO.INIT THEN
    FIFO.INIT		:= TRUE;
    FIFO.NW		:= 1;
    FIFO.NR		:= 1;
    FIFO.EMPTY	:= TRUE;
    FIFO.FULL		:= FALSE;
    FIFO.TOP		:= 128;
    FIFO.MAX_ID	:= BYTE#1;
  END_IF;

  IF ID = BYTE#00 THEN
    IF FIFO.ID < INT_TO_BYTE(FIFO.TOP) THEN
      ID := USINT_TO_BYTE(BYTE_TO_USINT(FIFO.ID) + USINT#1);
      FIFO.ID := ID ;

    ELSIF STATE < BYTE#200 THEN
      STATE := BYTE#255;
    RETURN;
    END_IF;
  END_IF;

  IF STATE = BYTE#1 AND NOT FIFO.FULL THEN
    tmp := _BYTE_TO_INT(ID);
    IF FIFO.Y[tmp] < FIFO.MAX_ID THEN
      FIFO.Y[tmp] := USINT_TO_BYTE(BYTE_TO_USINT(FIFO.Y[tmp]) + USINT#1);
      tmp := FIFO.NW;
      FIFO.X[tmp] := ID;
      IF FIFO.NW = FIFO.TOP THEN FIFO.NW := 1; ELSE FIFO.NW := FIFO.NW + 1; END_IF;
      FIFO.FULL := FIFO.NW = FIFO.NR;
    FIFO.EMPTY := FALSE;
      STATE := BYTE#2;
    END_IF;
  END_IF;

  IF STATE = BYTE#2 AND NOT FIFO.EMPTY THEN
    tmp := FIFO.NR;
    IF ID = FIFO.X[tmp] THEN
      STATE := BYTE#3;
    END_IF;
  END_IF;

  IF STATE = BYTE#4 AND NOT FIFO.EMPTY THEN

    tmp := FIFO.NR;
    IF ID = FIFO.X[tmp] THEN
      tmp := _BYTE_TO_INT(ID);
      FIFO.Y[tmp] := USINT_TO_BYTE(BYTE_TO_USINT(FIFO.Y[tmp]) - USINT#1);

      IF FIFO.NR = FIFO.TOP THEN FIFO.NR := 1; ELSE FIFO.NR := FIFO.NR + 1; END_IF;
      FIFO.EMPTY := FIFO.NR = FIFO.NW;
    FIFO.FULL := FALSE;
    END_IF;
    STATE := BYTE#5;
  END_IF;

END_FUNCTION_BLOCK

FUNCTION WORD_OF_BYTE:WORD
	VAR_INPUT
		B1 :	BYTE;
		B0 :	BYTE;
	END_VAR
	WORD_OF_BYTE := SHL(BYTE_TO_WORD(B1),8) OR BYTE_TO_WORD(B0);
END_FUNCTION

FUNCTION BIT_LOAD_W:WORD
	VAR_INPUT
		IN :	WORD;
		VAL :	BOOL;
		POS :	INT;
	END_VAR

	IF VAL THEN
		BIT_LOAD_W := in OR SHL(WORD#1,pos);
	ELSE
		BIT_LOAD_W := in AND (NOT SHL(WORD#1,pos));
	END_IF;
END_FUNCTION

FUNCTION_BLOCK MB_CLIENT_Block

	VAR_IN_OUT
		IP_C :	oscat_IP_C;
		S_BUF :	oscat_NETWORK_BUFFER_SHORT;
		R_BUF :	oscat_NETWORK_BUFFER_SHORT;
		DATA :	oscat_aW0_255;
	END_VAR

	VAR_INPUT
		DATA_SIZE :	INT;
		ENABLE :	BOOL;
		UDP :	BOOL;
		FC :	INT;
		UNIT_ID :	BYTE;
		R_ADDR :	INT;
		R_POINTS :	INT;
		R_DATA_ADR :	INT;
		R_DATA_BITPOS :	INT;
		W_ADDR :	INT;
		W_POINTS :	INT;
		W_DATA_ADR :	INT;
		W_DATA_BITPOS :	INT;
		DELAY :	TIME;
	END_VAR

	VAR_OUTPUT
		ERROR :	DWORD;
		BUSY :	BOOL;
	END_VAR

	VAR
		IP_STATE :	BYTE;
		IP_ID :	BYTE;
		IP_FIFO :	IP_FIFO_Block;
		mask :	DWORD;
		w_tmp :	WORD;
		idx1 :	INT;
		idx2 :	INT;
		stop :	INT;
		i :	INT;
		bit_pos :	INT;
		w_mask :	WORD;
		b_mask :	BYTE;
		count :	INT;
		state :	INT;
		Transaction_ID :	INT;
		Response :	INT;
		comp :	INT;
		TON_1 :	TON;
	END_VAR

	CASE state OF

	00:
		TON_1(IN:=ENABLE,PT:=DELAY);

		IF TON_1.Q OR DELAY = T#0s THEN
			TON_1(IN:=FALSE);
			state := 20;
			IP_STATE := BYTE#1;
		END_IF;

	20:
		IF IP_STATE = BYTE#3 THEN
			IP_C.C_PORT     := WORD#0;
			IP_C.C_IP       := DWORD#0;
			IP_C.C_MODE     := BOOL_TO_BYTE(UDP);
			IP_C.TIME_RESET := TRUE;
			IP_C.C_ENABLE   := TRUE;
			IP_C.R_OBSERVE  := TRUE;

			ERROR := DWORD#00;

			CASE FC OF

			1..2:
				IF R_POINTS <= 2000 THEN
					w_tmp := INT_TO_WORD(R_ADDR);
					S_BUF.BUFFER[08] := WORD_TO_BYTE(SHR(w_tmp,8));
					S_BUF.BUFFER[09] := WORD_TO_BYTE(w_tmp);
					w_tmp := INT_TO_WORD(R_POINTS);
					S_BUF.BUFFER[10] := WORD_TO_BYTE(SHR(w_tmp,8));
					S_BUF.BUFFER[11] := WORD_TO_BYTE(w_tmp);
					S_BUF.SIZE := UINT#12;
					Response :=	WORD_TO_INT(SHR(INT_TO_WORD(R_POINTS + 7),3));
					comp := 7;
				ELSE
					ERROR := DWORD#2;
				END_IF;
			3..4:
				IF R_POINTS <= 125 THEN
					w_tmp := INT_TO_WORD(R_ADDR);
					S_BUF.BUFFER[08] := WORD_TO_BYTE(SHR(w_tmp,8));
					S_BUF.BUFFER[09] := WORD_TO_BYTE(w_tmp);
					w_tmp := INT_TO_WORD(R_POINTS);
					S_BUF.BUFFER[10] := WORD_TO_BYTE(SHR(w_tmp,8));
					S_BUF.BUFFER[11] := WORD_TO_BYTE(w_tmp);

					S_BUF.SIZE := UINT#12;
					Response :=	WORD_TO_INT(SHL(w_tmp,1));
					comp := 7;
				ELSE
					ERROR := DWORD#2;
				END_IF;
			5:
				IF W_DATA_ADR <= DATA_SIZE THEN
					w_tmp := INT_TO_WORD(W_ADDR);
					S_BUF.BUFFER[08] := WORD_TO_BYTE(SHR(w_tmp,8));
					S_BUF.BUFFER[09] := WORD_TO_BYTE(w_tmp);
					S_BUF.BUFFER[10] := SEL((DATA[W_DATA_ADR] AND SHL(WORD#1,W_DATA_BITPOS))>WORD#00,BYTE#16#00,BYTE#16#FF);
					S_BUF.BUFFER[11] := BYTE#00;

					S_BUF.SIZE := UINT#12;
					Response :=	3;
					comp := 11;
				ELSE
					ERROR := DWORD#2;
				END_IF;
			6:
				IF W_DATA_ADR <= DATA_SIZE THEN
					w_tmp := INT_TO_WORD(W_ADDR);
					S_BUF.BUFFER[08] := WORD_TO_BYTE(SHR(w_tmp,8));
					S_BUF.BUFFER[09] := WORD_TO_BYTE(w_tmp);
					w_tmp := DATA[W_DATA_ADR];
					S_BUF.BUFFER[10] := WORD_TO_BYTE(SHR(w_tmp,8));
					S_BUF.BUFFER[11] := WORD_TO_BYTE(w_tmp);

					S_BUF.SIZE := UINT#12;
					Response :=	3;
					comp := 11;
				ELSE
					ERROR := DWORD#2;
				END_IF;
			15:
				IF (WORD_TO_INT(SHR(INT_TO_WORD(WORD_TO_INT(SHL(INT_TO_WORD(W_DATA_ADR),4)) + W_POINTS + W_DATA_BITPOS + 15),4)) <= DATA_SIZE) AND W_POINTS <= 1968 THEN
					w_tmp := INT_TO_WORD(W_ADDR);
					S_BUF.BUFFER[08] := WORD_TO_BYTE(SHR(w_tmp,8));
					S_BUF.BUFFER[09] := WORD_TO_BYTE(w_tmp);
					w_tmp := INT_TO_WORD(W_POINTS);
					S_BUF.BUFFER[10] := WORD_TO_BYTE(SHR(w_tmp,8));
					S_BUF.BUFFER[11] := WORD_TO_BYTE(w_tmp);
					S_BUF.BUFFER[12] := WORD_TO_BYTE(SHR(INT_TO_WORD(W_POINTS + 7),3));

					w_mask := SHL(WORD#1,W_DATA_BITPOS);
					bit_pos := 0;
					w_tmp := WORD#00;
					idx1 := 12;
					idx2 := W_DATA_ADR;
					FOR i := 1 TO W_POINTS DO
						w_tmp :=BIT_LOAD_W(w_tmp,(DATA[idx2] AND w_mask)>WORD#0,bit_pos);
						bit_pos := bit_pos + 1;
						IF bit_pos > 7 OR i=W_POINTS THEN
							bit_pos := 0;
							idx1 := idx1 + 1;
							S_BUF.BUFFER[idx1] := WORD_TO_BYTE(w_tmp);
							w_tmp := WORD#0;
						END_IF;
						w_mask := ROL(w_mask,1);
						IF w_mask = WORD#1 THEN
							idx2 := idx2 + 1;
						END_IF;
					END_FOR;
					S_BUF.SIZE := INT_TO_UINT(idx1+1);
					Response :=	3;
					comp := 11;
				ELSE
					ERROR := DWORD#2;
				END_IF;
			16:
				IF W_DATA_ADR + W_POINTS <= DATA_SIZE AND W_POINTS <= 123 THEN
					w_tmp := INT_TO_WORD(W_ADDR);
					S_BUF.BUFFER[08] := WORD_TO_BYTE(SHR(w_tmp,8));
					S_BUF.BUFFER[09] := WORD_TO_BYTE(w_tmp);
					w_tmp := INT_TO_WORD(W_POINTS);
					S_BUF.BUFFER[10] := WORD_TO_BYTE(SHR(w_tmp,8));
					S_BUF.BUFFER[11] := WORD_TO_BYTE(w_tmp);
					S_BUF.BUFFER[12] := SHL(S_BUF.BUFFER[11],1);

					idx1 := 11;
					count := W_DATA_ADR + W_POINTS - 1;
					FOR i := W_DATA_ADR TO count DO
						idx1 := idx1 + 2;
						idx2 := idx1 + 1;
						w_tmp := DATA[i];
						S_BUF.BUFFER[idx1] := WORD_TO_BYTE(SHR(w_tmp,8));
						S_BUF.BUFFER[idx2] := WORD_TO_BYTE(w_tmp);
					END_FOR;

					S_BUF.SIZE := INT_TO_UINT(idx2 + 1);
					Response := 3;
					comp := 11;
				ELSE
					ERROR := DWORD#2;
				END_IF;
			22:
				IF W_DATA_ADR + 2 <= DATA_SIZE THEN
					w_tmp := INT_TO_WORD(W_ADDR);
					S_BUF.BUFFER[08] := WORD_TO_BYTE(SHR(w_tmp,8));
					S_BUF.BUFFER[09] := WORD_TO_BYTE(w_tmp);
					idx1 := W_DATA_ADR;
					w_tmp := DATA[idx1];
					S_BUF.BUFFER[10] := WORD_TO_BYTE(SHR(w_tmp,8));
					S_BUF.BUFFER[11] := WORD_TO_BYTE(w_tmp);
					idx1 := idx1 +1;
					w_tmp := DATA[idx1];
					S_BUF.BUFFER[12] := WORD_TO_BYTE(SHR(w_tmp,8));
					S_BUF.BUFFER[13] := WORD_TO_BYTE(w_tmp);

					S_BUF.SIZE := UINT#14;
					Response :=	5;
					comp := 13;
				ELSE
					ERROR := DWORD#2;
				END_IF;
			23:
				IF W_DATA_ADR + W_POINTS <= DATA_SIZE AND W_POINTS <= 121 AND R_POINTS <= 125 THEN
					idx1 := 15;
					count := W_DATA_ADR + W_POINTS - 1;
					FOR i := W_DATA_ADR TO count DO
						idx1 := idx1 + 2;
						idx2 := idx1 + 1;
						w_tmp := DATA[i];
						S_BUF.BUFFER[idx1] := WORD_TO_BYTE(SHR(w_tmp,8));
						S_BUF.BUFFER[idx2] := WORD_TO_BYTE(w_tmp);
					END_FOR;

					w_tmp := INT_TO_WORD(W_ADDR);
					S_BUF.BUFFER[12] := WORD_TO_BYTE(SHR(w_tmp,8));
					S_BUF.BUFFER[13] := WORD_TO_BYTE(w_tmp);
					w_tmp := INT_TO_WORD(W_POINTS);
					S_BUF.BUFFER[14] := WORD_TO_BYTE(SHR(w_tmp,8));
					S_BUF.BUFFER[15] := WORD_TO_BYTE(w_tmp);
					S_BUF.BUFFER[16] := SHL(S_BUF.BUFFER[15],1);

					w_tmp := INT_TO_WORD(R_ADDR);
					S_BUF.BUFFER[08] := WORD_TO_BYTE(SHR(w_tmp,8));
					S_BUF.BUFFER[09] := WORD_TO_BYTE(w_tmp);
					w_tmp := INT_TO_WORD(R_POINTS);
					S_BUF.BUFFER[10] := WORD_TO_BYTE(SHR(w_tmp,8));
					S_BUF.BUFFER[11] := WORD_TO_BYTE(w_tmp);

					S_BUF.SIZE := INT_TO_UINT(idx2+1);
					Response :=	WORD_TO_INT(SHL(w_tmp,1));
					comp := 7;
				ELSE
					ERROR := DWORD#2;
				END_IF;

			ELSE
				ERROR := DWORD#00000001;
			END_CASE;

			IF ERROR = DWORD#00 THEN
				Transaction_ID := Transaction_ID + 1;
				w_tmp := UINT_TO_WORD(S_BUF.SIZE - UINT#6);
				S_BUF.BUFFER[0] := IP_ID;
				S_BUF.BUFFER[1] := INT_TO_BYTE(Transaction_ID);
				S_BUF.BUFFER[2] := BYTE#00;
				S_BUF.BUFFER[3] := BYTE#00;
				S_BUF.BUFFER[4] := WORD_TO_BYTE(SHR(w_tmp,8));
				S_BUF.BUFFER[5] := WORD_TO_BYTE(w_tmp);
				S_BUF.BUFFER[6] := UNIT_ID;
				S_BUF.BUFFER[7] := INT_TO_BYTE(FC);
				R_BUF.SIZE := UINT#0;
				state := 30;
			ELSE
				IP_STATE := BYTE#4;
				state := 00;
			END_IF;
		END_IF;

	30:
		IF IP_C.ERROR <> DWORD#00 THEN
			ERROR := IP_C.ERROR;
			IP_STATE := BYTE#4;
			state := 00;

		ELSIF S_BUF.SIZE = UINT#0 AND R_BUF.SIZE > UINT#0 THEN

			w_tmp := INT_TO_WORD(Response + 3);
			S_BUF.BUFFER[4] := WORD_TO_BYTE(SHR(w_tmp,8));
			S_BUF.BUFFER[5] := WORD_TO_BYTE(w_tmp);

			FOR i := 0 TO comp DO
				IF S_BUF.BUFFER[i] <> R_BUF.BUFFER[i] THEN EXIT; END_IF;
			END_FOR;

			IF R_BUF.SIZE >= UINT#9 AND R_BUF.BUFFER[7] > BYTE#128 THEN
				ERROR := BYTE_TO_DWORD(R_BUF.BUFFER[8]);
				IP_STATE := BYTE#4;
				state := 00;

			ELSIF R_BUF.SIZE = INT_TO_UINT(Response + 9) AND i > comp THEN
				mask := SHL(DWORD#1,FC);

				IF (mask AND DWORD#2#00000000_00000000_00000000_00000110) <> DWORD#0 THEN
					IF WORD_TO_INT(SHR(INT_TO_WORD(WORD_TO_INT(SHL(INT_TO_WORD(R_DATA_ADR),4)) + R_POINTS + R_DATA_BITPOS + 15),4)) <= DATA_SIZE THEN
						b_mask := BYTE#1;
						idx1 := 09;
						idx2 := R_DATA_ADR;
						bit_pos := R_DATA_BITPOS;
						FOR i := 1 TO R_POINTS DO
							DATA[idx2]:=BIT_LOAD_W(DATA[idx2],(R_BUF.BUFFER[idx1] AND b_mask)>BYTE#0,bit_pos);
							bit_pos := bit_pos + 1;
							IF bit_pos > 15 THEN
								idx2 := idx2 + 1;
								bit_pos := 0;
							END_IF;
							b_mask := ROL(b_mask,1);
							IF b_mask = BYTE#1 THEN
								idx1 := idx1 +1;
							END_IF;
						END_FOR;
					ELSE
						ERROR := DWORD#2;
					END_IF;

				ELSIF (mask AND DWORD#2#00000000_10000000_00000000_00011000) <> DWORD#0 THEN
					IF R_DATA_ADR + R_POINTS <= DATA_SIZE THEN
						stop := R_DATA_ADR + R_POINTS -1 ;
						idx1 := 07;
						FOR i := R_DATA_ADR TO stop DO
							idx1 := idx1 +2;
							idx2 := idx1 +1;
							DATA[i] := WORD_OF_BYTE(R_BUF.BUFFER[idx1],R_BUF.BUFFER[idx2]);
						END_FOR;
					ELSE
						ERROR := DWORD#2;
					END_IF;
				ELSIF (mask AND DWORD#2#11111111_00111110_01111111_10000001) > DWORD#0 THEN
					ERROR := DWORD#1;
				END_IF;
			ELSE
				ERROR := DWORD#3;
			END_IF;

			IP_STATE := BYTE#4;
			state := 00;
			R_BUF.SIZE := UINT#0;

		END_IF;

	END_CASE;

	IP_FIFO(FIFO:=IP_C.FIFO,STATE:=IP_STATE,ID:=IP_ID);
	IP_C.FIFO:=IP_FIFO.FIFO;
	IP_STATE := IP_FIFO.STATE;
	IP_ID:=IP_FIFO.ID;

	BUSY := IP_STATE = BYTE#3;

END_FUNCTION_BLOCK

PROGRAM program0
	VAR
		IP_C :	oscat_IP_C;
		S_BUF :	oscat_NETWORK_BUFFER_SHORT;
		R_BUF :	oscat_NETWORK_BUFFER_SHORT;
		DATA :	oscat_aW0_255;
		DATA_SIZE :	INT;
		ENABLE :	BOOL;
		UDP :	BOOL;
		FC :	INT;
		UNIT_ID :	BYTE;
		R_ADDR :	INT;
		R_POINTS :	INT;
		R_DATA_ADR :	INT;
		R_DATA_BITPOS :	INT;
		W_POINTS :	INT;
		W_DATA_ADR :	INT;
		W_DATA_BITPOS :	INT;
		DELAY :	TIME;
		ERROR :	DWORD;
		BUSY :	BOOL;

		func_block : MB_CLIENT_Block;
	END_VAR
	func_block.IP_C := IP_C;
	func_block.S_BUF := S_BUF;
	func_block.R_BUF := R_BUF;
	func_block.DATA := DATA;
	func_block.DATA_SIZE := DATA_SIZE;
	func_block.ENABLE := ENABLE;
	func_block.UDP := UDP;
	func_block.FC := FC;
	func_block.UNIT_ID := UNIT_ID;
	func_block.R_ADDR := R_ADDR;
	func_block.R_POINTS := R_POINTS;
	func_block.R_DATA_ADR := R_DATA_ADR;
	func_block.R_DATA_BITPOS := R_DATA_BITPOS;
	func_block.W_DATA_ADR := W_DATA_ADR;
	func_block.W_POINTS := W_POINTS;
	func_block.W_DATA_BITPOS := W_DATA_BITPOS;
	func_block.DELAY := DELAY;

	func_block();
  	IP_C  := func_block.IP_C;
	S_BUF  := func_block.S_BUF;
	R_BUF  := func_block.R_BUF;
	DATA  := func_block.DATA;
	ERROR  := func_block.ERROR;
	BUSY  := func_block.BUSY;

END_PROGRAM

CONFIGURATION Config0

	VAR_GLOBAL
		PLC_TICKS_PER_SEC :	INT;
		PLC_SYS_TICK_CNT :	DINT;
	END_VAR

  	RESOURCE Res0 ON PLC
    	TASK task0(INTERVAL := T#20ms,PRIORITY := 0);
    	PROGRAM instance0 WITH task0 : program0;
  	END_RESOURCE

END_CONFIGURATION
